# B&R Automation Studio project TD52 (part 43)

#### c_parCyclic.st
```iecst
(*******************************************************************************
CUSTOMIZED: c_par 			customized reserve parameters 1-200

This code is confidential and proprietary to the INNIO Company.
It may not be used in any form, or reproduced in any manner,
without written permission of the INNIO Company.
Copyright, INNIO Company, 2019

Customized modifications: -
------------------------

History:
-------
V3.20.0	02.03.2011 lettenb.	new, old default-settings removed
...
V4.00.0	08.05.2014 Zengerer ?hit? to int with optional factory default values
V4.02.0 24.06.2015 Zengerer cleanup
V4.04.0	20.06.2016 Weitzer	add reserve parameter 71..200
V4.11.0	31.01.2022 Zengerer	array preparation for import HMI Extensions 201..500

Instructions for use:
--------------------
- define customized use of reserve parameters here
- mark used channels here, to avoid duplicate usage withhin one customer project

AVOID HARDCODED Para.xxx VALUES!
You MAYBE want to enter SOME factory default values, but ONLY TO THE Para_FactoryDefault.xxx STRUCTURE!
By this way the parameter values in Para.xxx would stay acessible according to XT4 parameter management process.

***********************************************
further use for TP only!
***********************************************

Outstandings:
------------
	Para.iCtr_Mns_Options := REAL_TO_INT(Para.rCust_SparePara[72]) ;		ToDO: remove, when parameter gets availabel on VIS

*******************************************************************************)
PROGRAM _CYCLIC

	Para.rCust_SparePara[1]	;	(*MARK USAGE HERE, to avoid duplicate usage*)	(*  =   SPS_REZP1 *)
	OUT_CU.rCust_SparePara[1];	(*para values get copied to module OUT interface, to allow possible usage in other modules also. Edit other´s module .vvm accordingly, if needed. *)

	Para.rCust_SparePara[2]	; 													(*  =   SPS_REZP2 *)
	OUT_CU.rCust_SparePara[2];													(*  =	SPS_REZP2 *)

	Para.rCust_SparePara[3]	;  													(*  =	SPS_REZP3 *)
	OUT_CU.rCust_SparePara[3];													(*  =	SPS_REZP3 *)

	Para.rCust_SparePara[4]	;													(*  =   SPS_REZP4*)
	OUT_CU.rCust_SparePara[4];													(*  =	SPS_REZP4 *)

	Para.rCust_SparePara[5]	; 													(*  =   SPS_REZP5*)
	OUT_CU.rCust_SparePara[5];													(*  =	SPS_REZP5 *)

	Para.rCust_SparePara[6]	;  													(*  =	SPS_REZP6*)
	OUT_CU.rCust_SparePara[6];													(*  =	SPS_REZP6 *)

	Para.rCust_SparePara[7]	;  													(*  =	SPS_REZP7*)
	OUT_CU.rCust_SparePara[7] ;													(*  =	SPS_REZP7 *)

	Para.rCust_SparePara[8]	;   												(*  =	SPS_REZP8*)
	OUT_CU.rCust_SparePara[8] ;													(*  =	SPS_REZP8 *)

	Para.rCust_SparePara[9]		;  												(*  =	SPS_REZP9*)
	OUT_CU.rCust_SparePara[9] 	;												(*  =	SPS_REZP9 *)

	Para.rCust_SparePara[10]	;  												(*  =	SPS_REZP10*)
	OUT_CU.rCust_SparePara[10]	;												(*  =	SPS_REZP10 *)

	(*------------------------------------------------------------------*)
	Para.rCust_SparePara[11] 	;	(*  =	SPS_REZP11 *)
	OUT_CU.rCust_SparePara[11]	;	(*  =	SPS_REZP11 *)

	Para.rCust_SparePara[12]	;	(*  =	SPS_REZP12 *)
	OUT_CU.rCust_SparePara[12]	;	(*  =	SPS_REZP12 *)

	Para.rCust_SparePara[13]	;	(*  =	SPS_REZP13 *)
	OUT_CU.rCust_SparePara[13]	;	(*  =	SPS_REZP13 *)

	Para.rCust_SparePara[14]	;	(*  =	SPS_REZP14 *)
	OUT_CU.rCust_SparePara[14]	;	(*  =	SPS_REZP14 *)

	Para.rCust_SparePara[15]	;	(*  =	SPS_REZP15 *)
	OUT_CU.rCust_SparePara[15]	;	(*  =	SPS_REZP15 *)

	Para.rCust_SparePara[16]	;	(*  =	SPS_REZP16 *)
	OUT_CU.rCust_SparePara[16]	;	(*  =	SPS_REZP16 *)

	Para.rCust_SparePara[17]	;	(*  =	SPS_REZP17 *)
	OUT_CU.rCust_SparePara[17]	;	(*  =	SPS_REZP17 *)

	Para.rCust_SparePara[18]	;	(*  =	SPS_REZP18 *)
	OUT_CU.rCust_SparePara[18]	;	(*  =	SPS_REZP18 *)

	Para.rCust_SparePara[19]	;	(*  =	SPS_REZP19 *)
	OUT_CU.rCust_SparePara[19]	;	(*  =	SPS_REZP19 *)

	Para.rCust_SparePara[20]	;	(*  =	SPS_REZP20 *)
	OUT_CU.rCust_SparePara[20]	;	(*  =	SPS_REZP20 *)

	(*------------------------------------------------------------------*)
	Para.rCust_SparePara[21]	;	(*  =	SPS_REZP21*)
	OUT_CU.rCust_SparePara[21] ;	(*  =	SPS_REZP21; *)

	Para.rCust_SparePara[22]	;	(*  =	SPS_REZP22*)
	OUT_CU.rCust_SparePara[22] ;	(*  =	SPS_REZP22; *)

	Para.rCust_SparePara[23]	;	(*  =	SPS_REZP23*)
	OUT_CU.rCust_SparePara[23] ;	(*  =	SPS_REZP23; *)

	Para.rCust_SparePara[24]	;	(*  =	SPS_REZP24*)
	OUT_CU.rCust_SparePara[24] ;	(*  =	SPS_REZP24; *)

	Para.rCust_SparePara[25]	;	(*  =	SPS_REZP25*)
	OUT_CU.rCust_SparePara[25] ;	(*  =	SPS_REZP25; *)

	Para.rCust_SparePara[26]	;	(*  =	SPS_REZP26*)
	OUT_CU.rCust_SparePara[26] ;	(*  =	SPS_REZP26; *)

	Para.rCust_SparePara[27]	;	(*  =	SPS_REZP27*)
	OUT_CU.rCust_SparePara[27] ;	(*  =	SPS_REZP27; *)

	Para.rCust_SparePara[28]	;	(*  =	SPS_REZP28*)
	OUT_CU.rCust_SparePara[28] ;	(*  =	SPS_REZP28; *)

	Para.rCust_SparePara[29]	;	(*  =	SPS_REZP29*)
	OUT_CU.rCust_SparePara[29] ;	(*  =	SPS_REZP29; *)

	OUT_CU.rCust_SparePara[30] ;	(*  =	SPS_REZP30; *)

	(*------------------------------------------------------------------*)
	Para.rCust_SparePara[31]	;	(*  =	SPS_REZP31*)
	OUT_CU.rCust_SparePara[31] ;	(*  =	SPS_REZP31; *)

	Para.rCust_SparePara[32]	;	(*  =	SPS_REZP32*)
	OUT_CU.rCust_SparePara[32] ;	(*  =	SPS_REZP32; *)

	Para.rCust_SparePara[33]	;	(*  =	SPS_REZP33*)
	OUT_CU.rCust_SparePara[33] ;	(*  =	SPS_REZP33; *)

	Para.rCust_SparePara[34]	;	(*  =	SPS_REZP34*)
	OUT_CU.rCust_SparePara[34] ;	(*  =	SPS_REZP34; *)

	Para.rCust_SparePara[35]	;	(*  =	SPS_REZP35*)
	OUT_CU.rCust_SparePara[35] ;	(*  =	SPS_REZP35; *)

	Para.rCust_SparePara[36]	;	(*  =	SPS_REZP36*)
	OUT_CU.rCust_SparePara[36] ;	(*  =	SPS_REZP36; *)

	Para.rCust_SparePara[37]	;	(*  =	SPS_REZP37*)
	OUT_CU.rCust_SparePara[37] ;	(*  =	SPS_REZP37; *)

	Para.rCust_SparePara[38]	;	(*  =	SPS_REZP38*)
	OUT_CU.rCust_SparePara[38] ;	(*  =	SPS_REZP38; *)

	Para.rCust_SparePara[39]	;	(*  =	SPS_REZP39*)
	OUT_CU.rCust_SparePara[39] ;	(*  =	SPS_REZP39; *)

	Para.rCust_SparePara[40]	;	(*  =	SPS_REZP40*)
	OUT_CU.rCust_SparePara[40] ;	(*  =	SPS_REZP40; *)

	(*------------------------------------------------------------------*)
	Para.rCust_SparePara[41]	;	(*  =	SPS_REZP41*)
	OUT_CU.rCust_SparePara[41] ;	(*  =	SPS_REZP41; *)

	Para.rCust_SparePara[42]	;	(*  =	SPS_REZP42*)
	OUT_CU.rCust_SparePara[42] ;	(*  =	SPS_REZP42; *)

	Para.rCust_SparePara[43]	;	(*  =	SPS_REZP43*)
	OUT_CU.rCust_SparePara[43] ;	(*  =	SPS_REZP43; *)

	Para.rCust_SparePara[44]	;	(*  =	SPS_REZP44*)
	OUT_CU.rCust_SparePara[44] ;	(*  =	SPS_REZP44; *)

	Para.rCust_SparePara[45]	;	(*  =	SPS_REZP45*)
	OUT_CU.rCust_SparePara[45] ;	(*  =	SPS_REZP45; *)

	Para.rCust_SparePara[46]	;	(*  =	SPS_REZP46*)
	OUT_CU.rCust_SparePara[46] ;	(*  =	SPS_REZP46; *)

	Para.rCust_SparePara[47]	;	(*  =	SPS_REZP47*)
	OUT_CU.rCust_SparePara[47] ;	(*  =	SPS_REZP47; *)

	Para.rCust_SparePara[48]	;	(*  =	SPS_REZP48*)
	OUT_CU.rCust_SparePara[48] ;	(*  =	SPS_REZP48; *)

	Para.rCust_SparePara[49]	;	(*  =	SPS_REZP49*)
	OUT_CU.rCust_SparePara[49] ;	(*  =	SPS_REZP49; *)

	Para.rCust_SparePara[50]	;	(*  =	SPS_REZP50*)
	OUT_CU.rCust_SparePara[50] ;	(*  =	SPS_REZP50; *)

	(*------------------------------------------------------------------*)
	Para.rCust_SparePara[51]	;	(*  =	SPS_REZP51*)
	OUT_CU.rCust_SparePara[51] ;	(*  =	SPS_REZP51; *)

	Para.rCust_SparePara[52]	;	(*  =	SPS_REZP52*)
	OUT_CU.rCust_SparePara[52] ;	(*  =	SPS_REZP52; *)

	Para.rCust_SparePara[53]	;	(*  =	SPS_REZP53*)
	OUT_CU.rCust_SparePara[53] ;	(*  =	SPS_REZP53; *)

	Para.rCust_SparePara[54]	;	(*  =	SPS_REZP54*)
	OUT_CU.rCust_SparePara[54] ;	(*  =	SPS_REZP54; *)

	Para.rCust_SparePara[55]	;	(*  =	SPS_REZP55*)
	OUT_CU.rCust_SparePara[55] ;	(*  =	SPS_REZP55; *)

	Para.rCust_SparePara[56]	;	(*  =	SPS_REZP56*)
	OUT_CU.rCust_SparePara[56] ;	(*  =	SPS_REZP56; *)

	Para.rCust_SparePara[57]	;	(*  =	SPS_REZP57*)
	OUT_CU.rCust_SparePara[57] ;	(*  =	SPS_REZP57; *)

	Para.rCust_SparePara[58]	;	(*  =	SPS_REZP58*)
	OUT_CU.rCust_SparePara[58] ;	(*  =	SPS_REZP58; *)

	Para.rCust_SparePara[59]	;	(*  =	SPS_REZP59*)
	OUT_CU.rCust_SparePara[59] ;	(*  =	SPS_REZP59; *)

	Para.rCust_SparePara[60]	;	(*  =	SPS_REZP60*)
	OUT_CU.rCust_SparePara[60] ;	(*  =	SPS_REZP60; *)

	(*------------------------------------------------------------------*)
	Para.rCust_SparePara[61]	;	(*  =	SPS_REZP61*)
	OUT_CU.rCust_SparePara[61] ;	(* = 	ssResPara61 *)

	Para.rCust_SparePara[62]	;	(*  =	SPS_REZP62*)
	OUT_CU.rCust_SparePara[62] ;	(* = 	ssResPara62 *)

	Para.rCust_SparePara[63]	;	(*  =	SPS_REZP63*)
	OUT_CU.rCust_SparePara[63] ;	(* = 	ssResPara63 *)

	Para.rCust_SparePara[64]	;	(*  =	SPS_REZP64*)
	OUT_CU.rCust_SparePara[64] ;	(* = 	ssResPara64 *)

	Para.rCust_SparePara[65]	;	(*  =	SPS_REZP65*)
	OUT_CU.rCust_SparePara[65] ;	(* = 	ssResPara65 *)

	Para.rCust_SparePara[66]	;	(*  =	SPS_REZP66*)
	OUT_CU.rCust_SparePara[66] ;	(* = 	ssResPara66 *)

	Para.rCust_SparePara[67]	;	(*  =	SPS_REZP67*)
	OUT_CU.rCust_SparePara[67] ;	(* = 	ssResPara67 *)

	Para.rCust_SparePara[68]	;	(*  =	SPS_REZP68*)
	OUT_CU.rCust_SparePara[68] ;	(* = 	ssResPara68 *)

	Para.rCust_SparePara[69]	;	(*  =	SPS_REZP69 *)
	OUT_CU.rCust_SparePara[69] ;	(* = 	ssResPara69 *)

	Para.rCust_SparePara[70]	;	(*  =	SPS_REZP70 *)
	OUT_CU.rCust_SparePara[70] ;	(* = 	ssResPara70 *)

	(*---------------------------------------------------------------------------------------*)
	(* END OF PRECONFIGURED VISUALISATION DATA POINS on standard engines, up to Vis Rev. 4.x *)
	(*---------------------------------------------------------------------------------------*)
	Para.rCust_SparePara[71];		(*  = SPS_REZP	71	***USED*** *)
	OUT_CU.rCust_SparePara[71];		(*  = ssResPara	71	*)

	Para.rCust_SparePara[72];		(*  = SPS_REZP	72  ***USED*** *)
	OUT_CU.rCust_SparePara[72];		(*  = ssResPara	72	*)

	Para.rCust_SparePara[73];		(*  = SPS_REZP	73	***USED*** *)
	OUT_CU.rCust_SparePara[73];		(*  = ssResPara	73	*)

	Para.rCust_SparePara[74];		(*  = SPS_REZP	74	*)
	OUT_CU.rCust_SparePara[74];		(*  = ssResPara	74	*)

	Para.rCust_SparePara[75];		(*  = SPS_REZP	75	*)
	OUT_CU.rCust_SparePara[75];		(*  = ssResPara	75	*)

	Para.rCust_SparePara[76];		(*  = SPS_REZP	76	*)
	OUT_CU.rCust_SparePara[76];		(*  = ssResPara	76	*)

	Para.rCust_SparePara[77];		(*  = SPS_REZP	77	*)
	OUT_CU.rCust_SparePara[77];		(*  = ssResPara	77	*)

	Para.rCust_SparePara[78];		(*  = SPS_REZP	78	*)
	OUT_CU.rCust_SparePara[78];		(*  = ssResPara	78	*)

	Para.rCust_SparePara[79];		(*  = SPS_REZP	79	*)
	OUT_CU.rCust_SparePara[79];		(*  = ssResPara	79	*)

	Para.rCust_SparePara[80];		(*  = SPS_REZP	80	*)
	OUT_CU.rCust_SparePara[80];		(*  = ssResPara	80	*)

	(*------------------------------------------------------------------*)
	Para.rCust_SparePara[81];		(*  = SPS_REZP	81	*)
	OUT_CU.rCust_SparePara[81];		(*  = ssResPara	81	*)

	Para.rCust_SparePara[82];		(*  = SPS_REZP	82	*)
	OUT_CU.rCust_SparePara[82];		(*  = ssResPara	82	*)

	Para.rCust_SparePara[83];		(*  = SPS_REZP	83	*)
	OUT_CU.rCust_SparePara[83];		(*  = ssResPara	83	*)

	Para.rCust_SparePara[84];		(*  = SPS_REZP	84	*)
	OUT_CU.rCust_SparePara[84];		(*  = ssResPara	84	*)

	Para.rCust_SparePara[85];		(*  = SPS_REZP	85	*)
	OUT_CU.rCust_SparePara[85];		(*  = ssResPara	85	*)

	Para.rCust_SparePara[86];		(*  = SPS_REZP	86	*)
	OUT_CU.rCust_SparePara[86];		(*  = ssResPara	86	*)

	Para.rCust_SparePara[87];		(*  = SPS_REZP	87	*)
	OUT_CU.rCust_SparePara[87];		(*  = ssResPara	87	*)

	Para.rCust_SparePara[88];		(*  = SPS_REZP	88	*)
	OUT_CU.rCust_SparePara[88];		(*  = ssResPara	88	*)

	Para.rCust_SparePara[89];		(*  = SPS_REZP	89	*)
	OUT_CU.rCust_SparePara[89];		(*  = ssResPara	89	*)

	Para.rCust_SparePara[90];		(*  = SPS_REZP	90	*)
	OUT_CU.rCust_SparePara[90];		(*  = ssResPara	90	*)

	(*------------------------------------------------------------------*)
	Para.rCust_SparePara[91];		(*  = SPS_REZP	91	*)
	OUT_CU.rCust_SparePara[91];		(*  = ssResPara	91	*)

	Para.rCust_SparePara[92];		(*  = SPS_REZP	92	*)
	OUT_CU.rCust_SparePara[92];		(*  = ssResPara	92	*)

	Para.rCust_SparePara[93];		(*  = SPS_REZP	93	*)
	OUT_CU.rCust_SparePara[93];		(*  = ssResPara	93	*)

	Para.rCust_SparePara[94];		(*  = SPS_REZP	94	*)
	OUT_CU.rCust_SparePara[94];		(*  = ssResPara	94	*)

	Para.rCust_SparePara[95];		(*  = SPS_REZP	95	*)
	OUT_CU.rCust_SparePara[95];		(*  = ssResPara	95	*)

	Para.rCust_SparePara[96];		(*  = SPS_REZP	96	*)
	OUT_CU.rCust_SparePara[96];		(*  = ssResPara	96	*)

	Para.rCust_SparePara[97];		(*  = SPS_REZP	97	*)
	OUT_CU.rCust_SparePara[97];		(*  = ssResPara	97	*)

	Para.rCust_SparePara[98];		(*  = SPS_REZP	98	*)
	OUT_CU.rCust_SparePara[98];		(*  = ssResPara	98	*)

	Para.rCust_SparePara[99];		(*  = SPS_REZP	99	*)
	OUT_CU.rCust_SparePara[99];		(*  = ssResPara	99	*)

	Para.rCust_SparePara[100];		(*  = SPS_REZP	100	*)
	OUT_CU.rCust_SparePara[100];	(*  = ssResPara	100	*)

	(*------------------------------------------------------------------*)
	Para.rCust_SparePara[101];		(*  = SPS_REZP	101	*)
	OUT_CU.rCust_SparePara[101];	(*  = ssResPara	101	*)

	Para.rCust_SparePara[102];		(*  = SPS_REZP	102	*)
	OUT_CU.rCust_SparePara[102];	(*  = ssResPara	102	*)

	Para.rCust_SparePara[103];		(*  = SPS_REZP	103	*)
	OUT_CU.rCust_SparePara[103];	(*  = ssResPara	103	*)

	Para.rCust_SparePara[104];		(*  = SPS_REZP	104	*)
	OUT_CU.rCust_SparePara[104];	(*  = ssResPara	104	*)

	Para.rCust_SparePara[105];		(*  = SPS_REZP	105	*)
	OUT_CU.rCust_SparePara[105];	(*  = ssResPara	105	*)

	Para.rCust_SparePara[106];		(*  = SPS_REZP	106	*)
	OUT_CU.rCust_SparePara[106];	(*  = ssResPara	106	*)

	Para.rCust_SparePara[107];		(*  = SPS_REZP	107	*)
	OUT_CU.rCust_SparePara[107];	(*  = ssResPara	107	*)

	Para.rCust_SparePara[108];		(*  = SPS_REZP	108	*)
	OUT_CU.rCust_SparePara[108];	(*  = ssResPara	108	*)

	Para.rCust_SparePara[109];		(*  = SPS_REZP	109	*)
	OUT_CU.rCust_SparePara[109];	(*  = ssResPara	109	*)

	Para.rCust_SparePara[110];		(*  = SPS_REZP	110	*)
	OUT_CU.rCust_SparePara[110];	(*  = ssResPara	110	*)

	(*------------------------------------------------------------------*)
	Para.rCust_SparePara[111];		(*  = SPS_REZP	111	*)
	OUT_CU.rCust_SparePara[111];	(*  = ssResPara	111	*)

	Para.rCust_SparePara[112];		(*  = SPS_REZP	112	*)
	OUT_CU.rCust_SparePara[112];	(*  = ssResPara	112	*)

	Para.rCust_SparePara[113];		(*  = SPS_REZP	113	*)
	OUT_CU.rCust_SparePara[113];	(*  = ssResPara	113	*)

	Para.rCust_SparePara[114];		(*  = SPS_REZP	114	*)
	OUT_CU.rCust_SparePara[114];	(*  = ssResPara	114	*)

	Para.rCust_SparePara[115];		(*  = SPS_REZP	115	*)
	OUT_CU.rCust_SparePara[115];	(*  = ssResPara	115	*)

	Para.rCust_SparePara[116];		(*  = SPS_REZP	116	*)
	OUT_CU.rCust_SparePara[116];	(*  = ssResPara	116	*)

	Para.rCust_SparePara[117];		(*  = SPS_REZP	117	*)
	OUT_CU.rCust_SparePara[117];	(*  = ssResPara	117	*)

	Para.rCust_SparePara[118];		(*  = SPS_REZP	118	*)
	OUT_CU.rCust_SparePara[118];	(*  = ssResPara	118	*)

	Para.rCust_SparePara[119];		(*  = SPS_REZP	119	*)
	OUT_CU.rCust_SparePara[119];	(*  = ssResPara	119	*)

	Para.rCust_SparePara[120];		(*  = SPS_REZP	120	*)
	OUT_CU.rCust_SparePara[120];	(*  = ssResPara	120	*)

	(*------------------------------------------------------------------*)
	Para.rCust_SparePara[121];		(*  = SPS_REZP	121	*)
	OUT_CU.rCust_SparePara[121];	(*  = ssResPara	121	*)

	Para.rCust_SparePara[122];		(*  = SPS_REZP	122	*)
	OUT_CU.rCust_SparePara[122];	(*  = ssResPara	122	*)

	Para.rCust_SparePara[123];		(*  = SPS_REZP	123	*)
	OUT_CU.rCust_SparePara[123];	(*  = ssResPara	123	*)

	Para.rCust_SparePara[124];		(*  = SPS_REZP	124	*)
	OUT_CU.rCust_SparePara[124];	(*  = ssResPara	124	*)

	Para.rCust_SparePara[125];		(*  = SPS_REZP	125	*)
	OUT_CU.rCust_SparePara[125];	(*  = ssResPara	125	*)

	Para.rCust_SparePara[126];		(*  = SPS_REZP	126	*)
	OUT_CU.rCust_SparePara[126];	(*  = ssResPara	126	*)

	Para.rCust_SparePara[127];		(*  = SPS_REZP	127	*)
	OUT_CU.rCust_SparePara[127];	(*  = ssResPara	127	*)

	Para.rCust_SparePara[128];		(*  = SPS_REZP	128	*)
	OUT_CU.rCust_SparePara[128];	(*  = ssResPara	128	*)

	Para.rCust_SparePara[129];		(*  = SPS_REZP	129	*)
	OUT_CU.rCust_SparePara[129];	(*  = ssResPara	129	*)

	Para.rCust_SparePara[130];		(*  = SPS_REZP	130	*)
	OUT_CU.rCust_SparePara[130];	(*  = ssResPara	130	*)

	(*------------------------------------------------------------------*)
	Para.rCust_SparePara[131];		(*  = SPS_REZP	131	*)
	OUT_CU.rCust_SparePara[131];	(*  = ssResPara	131	*)

	Para.rCust_SparePara[132];		(*  = SPS_REZP	132	*)
	OUT_CU.rCust_SparePara[132];	(*  = ssResPara	132	*)

	Para.rCust_SparePara[133];		(*  = SPS_REZP	133	*)
	OUT_CU.rCust_SparePara[133];	(*  = ssResPara	133	*)

	Para.rCust_SparePara[134];		(*  = SPS_REZP	134	*)
	OUT_CU.rCust_SparePara[134];	(*  = ssResPara	134	*)

	Para.rCust_SparePara[135];		(*  = SPS_REZP	135	*)
	OUT_CU.rCust_SparePara[135];	(*  = ssResPara	135	*)

	Para.rCust_SparePara[136];		(*  = SPS_REZP	136	*)
	OUT_CU.rCust_SparePara[136];	(*  = ssResPara	136	*)

	Para.rCust_SparePara[137];		(*  = SPS_REZP	137	*)
	OUT_CU.rCust_SparePara[137];	(*  = ssResPara	137	*)

	Para.rCust_SparePara[138];		(*  = SPS_REZP	138	*)
	OUT_CU.rCust_SparePara[138];	(*  = ssResPara	138	*)

	Para.rCust_SparePara[139];		(*  = SPS_REZP	139	*)
	OUT_CU.rCust_SparePara[139];	(*  = ssResPara	139	*)

	Para.rCust_SparePara[140];		(*  = SPS_REZP	140	*)
	OUT_CU.rCust_SparePara[140];	(*  = ssResPara	140	*)

	(*------------------------------------------------------------------*)
	Para.rCust_SparePara[141];		(*  = SPS_REZP	141	*)
	OUT_CU.rCust_SparePara[141];	(*  = ssResPara	141	*)

	Para.rCust_SparePara[142];		(*  = SPS_REZP	142	*)
	OUT_CU.rCust_SparePara[142];	(*  = ssResPara	142	*)

	Para.rCust_SparePara[143];		(*  = SPS_REZP	143	*)
	OUT_CU.rCust_SparePara[143];	(*  = ssResPara	143	*)

	Para.rCust_SparePara[144];		(*  = SPS_REZP	144	*)
	OUT_CU.rCust_SparePara[144];	(*  = ssResPara	144	*)

	Para.rCust_SparePara[145];		(*  = SPS_REZP	145	*)
	OUT_CU.rCust_SparePara[145];	(*  = ssResPara	145	*)

	Para.rCust_SparePara[146];		(*  = SPS_REZP	146	*)
	OUT_CU.rCust_SparePara[146];	(*  = ssResPara	146	*)

	Para.rCust_SparePara[147];		(*  = SPS_REZP	147	*)
	OUT_CU.rCust_SparePara[147];	(*  = ssResPara	147	*)

	Para.rCust_SparePara[148];		(*  = SPS_REZP	148	*)
	OUT_CU.rCust_SparePara[148];	(*  = ssResPara	148	*)

	Para.rCust_SparePara[149];		(*  = SPS_REZP	149	*)
	OUT_CU.rCust_SparePara[149];	(*  = ssResPara	149	*)

	Para.rCust_SparePara[150];		(*  = SPS_REZP	150	*)
	OUT_CU.rCust_SparePara[150];	(*  = ssResPara	150	*)

	(*------------------------------------------------------------------*)
	Para.rCust_SparePara[151];		(*  = SPS_REZP	151	*)
	OUT_CU.rCust_SparePara[151];	(*  = ssResPara	151	*)

	Para.rCust_SparePara[152];		(*  = SPS_REZP	152	*)
	OUT_CU.rCust_SparePara[152];	(*  = ssResPara	152	*)

	Para.rCust_SparePara[153];		(*  = SPS_REZP	153	*)
	OUT_CU.rCust_SparePara[153];	(*  = ssResPara	153	*)

	Para.rCust_SparePara[154];		(*  = SPS_REZP	154	*)
	OUT_CU.rCust_SparePara[154];	(*  = ssResPara	154	*)

	Para.rCust_SparePara[155];		(*  = SPS_REZP	155	*)
	OUT_CU.rCust_SparePara[155];	(*  = ssResPara	155	*)

	Para.rCust_SparePara[156];		(*  = SPS_REZP	156	*)
	OUT_CU.rCust_SparePara[156];	(*  = ssResPara	156	*)

	Para.rCust_SparePara[157];		(*  = SPS_REZP	157	*)
	OUT_CU.rCust_SparePara[157];	(*  = ssResPara	157	*)

	Para.rCust_SparePara[158];		(*  = SPS_REZP	158	*)
	OUT_CU.rCust_SparePara[158];	(*  = ssResPara	158	*)

	Para.rCust_SparePara[159];		(*  = SPS_REZP	159	*)
	OUT_CU.rCust_SparePara[159];	(*  = ssResPara	159	*)

	Para.rCust_SparePara[160];		(*  = SPS_REZP	160	*)
	OUT_CU.rCust_SparePara[160];	(*  = ssResPara	160	*)

	(*------------------------------------------------------------------*)
	Para.rCust_SparePara[161];		(*  = SPS_REZP	161	*)
	OUT_CU.rCust_SparePara[161];	(*  = ssResPara	161	*)

	Para.rCust_SparePara[162];		(*  = SPS_REZP	162	*)
	OUT_CU.rCust_SparePara[162];	(*  = ssResPara	162	*)

	Para.rCust_SparePara[163];		(*  = SPS_REZP	163	*)
	OUT_CU.rCust_SparePara[163];	(*  = ssResPara	163	*)

	Para.rCust_SparePara[164];		(*  = SPS_REZP	164	*)
	OUT_CU.rCust_SparePara[164];	(*  = ssResPara	164	*)

	Para.rCust_SparePara[165];		(*  = SPS_REZP	165	*)
	OUT_CU.rCust_SparePara[165];	(*  = ssResPara	165	*)

	Para.rCust_SparePara[166];		(*  = SPS_REZP	166	*)
	OUT_CU.rCust_SparePara[166];	(*  = ssResPara	166	*)

	Para.rCust_SparePara[167];		(*  = SPS_REZP	167	*)
	OUT_CU.rCust_SparePara[167];	(*  = ssResPara	167	*)

	Para.rCust_SparePara[168];		(*  = SPS_REZP	168	*)
	OUT_CU.rCust_SparePara[168];	(*  = ssResPara	168	*)

	Para.rCust_SparePara[169];		(*  = SPS_REZP	169	*)
	OUT_CU.rCust_SparePara[169];	(*  = ssResPara	169	*)

	Para.rCust_SparePara[170];		(*  = SPS_REZP	170	*)
	OUT_CU.rCust_SparePara[170];	(*  = ssResPara	170	*)

	(*------------------------------------------------------------------*)
	Para.rCust_SparePara[171];		(*  = SPS_REZP	171	*)
	OUT_CU.rCust_SparePara[171];	(*  = ssResPara	171	*)

	Para.rCust_SparePara[172];		(*  = SPS_REZP	172	*)
	OUT_CU.rCust_SparePara[172];	(*  = ssResPara	172	*)

	Para.rCust_SparePara[173];		(*  = SPS_REZP	173	*)
	OUT_CU.rCust_SparePara[173];	(*  = ssResPara	173	*)

	Para.rCust_SparePara[174];		(*  = SPS_REZP	174	*)
	OUT_CU.rCust_SparePara[174];	(*  = ssResPara	174	*)

	Para.rCust_SparePara[175];		(*  = SPS_REZP	175	*)
	OUT_CU.rCust_SparePara[175];	(*  = ssResPara	175	*)

	Para.rCust_SparePara[176];		(*  = SPS_REZP	176	*)
	OUT_CU.rCust_SparePara[176];	(*  = ssResPara	176	*)

	Para.rCust_SparePara[177];		(*  = SPS_REZP	177	*)
	OUT_CU.rCust_SparePara[177];	(*  = ssResPara	177	*)

	Para.rCust_SparePara[178];		(*  = SPS_REZP	178	*)
	OUT_CU.rCust_SparePara[178];	(*  = ssResPara	178	*)

	Para.rCust_SparePara[179];		(*  = SPS_REZP	179	*)
	OUT_CU.rCust_SparePara[179];	(*  = ssResPara	179	*)

	Para.rCust_SparePara[180];		(*  = SPS_REZP	180	*)
	OUT_CU.rCust_SparePara[180];	(*  = ssResPara	180	*)

	(*------------------------------------------------------------------*)
	Para.rCust_SparePara[181];		(*  = SPS_REZP	181	*)
	OUT_CU.rCust_SparePara[181];	(*  = ssResPara	181	*)

	Para.rCust_SparePara[182];		(*  = SPS_REZP	182	*)
	OUT_CU.rCust_SparePara[182];	(*  = ssResPara	182	*)

	Para.rCust_SparePara[183];		(*  = SPS_REZP	183	*)
	OUT_CU.rCust_SparePara[183];	(*  = ssResPara	183	*)

	Para.rCust_SparePara[184];		(*  = SPS_REZP	184	*)
	OUT_CU.rCust_SparePara[184];	(*  = ssResPara	184	*)

	Para.rCust_SparePara[185];		(*  = SPS_REZP	185	*)
	OUT_CU.rCust_SparePara[185];	(*  = ssResPara	185	*)

	Para.rCust_SparePara[186];		(*  = SPS_REZP	186	*)
	OUT_CU.rCust_SparePara[186];	(*  = ssResPara	186	*)

	Para.rCust_SparePara[187];		(*  = SPS_REZP	187	*)
	OUT_CU.rCust_SparePara[187];	(*  = ssResPara	187	*)

	Para.rCust_SparePara[188];		(*  = SPS_REZP	188	*)
	OUT_CU.rCust_SparePara[188];	(*  = ssResPara	188	*)

	Para.rCust_SparePara[189];		(*  = SPS_REZP	189	*)
	OUT_CU.rCust_SparePara[189];	(*  = ssResPara	189	*)

	Para.rCust_SparePara[190];		(*  = SPS_REZP	190	*)
	OUT_CU.rCust_SparePara[190];	(*  = ssResPara	190	*)

	(*------------------------------------------------------------------*)
	Para.rCust_SparePara[191];		(*  = SPS_REZP	191	*)
	OUT_CU.rCust_SparePara[191];	(*  = ssResPara	191	*)

	Para.rCust_SparePara[192];		(*  = SPS_REZP	192	*)
	OUT_CU.rCust_SparePara[192];	(*  = ssResPara	192	*)

	Para.rCust_SparePara[193];		(*  = SPS_REZP	193	*)
	OUT_CU.rCust_SparePara[193];	(*  = ssResPara	193	*)

	Para.rCust_SparePara[194];		(*  = SPS_REZP	194	*)
	OUT_CU.rCust_SparePara[194];	(*  = ssResPara	194	*)

	Para.rCust_SparePara[195];		(*  = SPS_REZP	195	*)
	OUT_CU.rCust_SparePara[195];	(*  = ssResPara	195	*)

	Para.rCust_SparePara[196];		(*  = SPS_REZP	196	*)
	OUT_CU.rCust_SparePara[196];	(*  = ssResPara	196	*)

	Para.rCust_SparePara[197];		(*  = SPS_REZP	197	*)
	OUT_CU.rCust_SparePara[197];	(*  = ssResPara	197	*)

	Para.rCust_SparePara[198];		(*  = SPS_REZP	198	*)
	OUT_CU.rCust_SparePara[198];	(*  = ssResPara	198	*)

	Para.rCust_SparePara[199];		(*  = SPS_REZP	199	*)
	OUT_CU.rCust_SparePara[199];	(*  = ssResPara	199	*)

	Para.rCust_SparePara[200];		(*  = SPS_REZP	200	*)
	OUT_CU.rCust_SparePara[200];	(*  = ssResPara	200	*)

	(*------------------------------------------------------------------*)

	(***********************************************
	END OF CONFIGURATION AREA
	***********************************************)
	(* NO CHANGES BEJOND THIS LINE! *)

//	OUT_CU.rCust_SparePara := 		Para.rCust_SparePara     ;	(* DONT DO THIS ANY MORE since different array size is possible with HMI Extention import in V4.11  *)
	iOut_SparePara_Size := SIZEOF(OUT_CU.rCust_SparePara)/ SIZEOF(OUT_CU.rCust_SparePara[0]) -1 ;
	FOR n := 0 TO iOut_SparePara_Size DO
		OUT_CU.rCust_SparePara[n] := 		Para.rCust_SparePara[n]     ;	(* Copy all parameter values to Module OUT interface for possible reuse in other modules  *)
	END_FOR

END_PROGRAM
```

#### c_par.var
```iecst
VAR
	iOut_SparePara_Size : UDINT := 0;
	n : UDINT := 0;
END_VAR
```

### Program Logical/Customized/c_ctr (IEC, version 4.11.0) - Interface connection for  customizable controllers

#### c_ctrCyclic.st - Cyclic code
```iecst
(*******************************************************************************
CUSTOMIZED: c_ctr 		reserve controller handling (cyclic)

This code is confidential AND proprietary to the INNIO Company.
It may NOT be used in any form, or reproduced in any manner,
without written permission of the INNIO Company.
Copyright, INNIO Company, 2022

Customized modifications: -
------------------------

History:
-------
		23.05.2012	Zengerer	generated, new
V4.02	09.09.2015	Zengerer	cleanup, prototype entry FOR documentation comments
V4.04	20.06.2016	Weitzer		add controller 41 .. 45
V4.05	23.01.2018	Perktold	added option for humitity control with ctr. 2
V4.11	27.01.2022	Perktold	impemented plant controller upgrade (2nd W_set, Gain Scheduling, Retrigger, cust. Ymin/max)
		31.01.2022	zengerer	extended controller items 41-45 ONLY FOR USE WITH HMI Extension Package!

Instructions FOR use:
--------------------
-
Outstandings:
------------
- ENTFERNEN: IF NOT bEnableTestBench THEN   (*NUR FÜR TPSS- Prüfstand...

*******************************************************************************)

PROGRAM _CYCLIC
																																		//	IF NOT bEnableTestBench THEN   (*Bit bEnableTestBench NUR FÜR TP- Prüfstand aktivieren*)

	(* customizable controller X 		*** PROTOTYPE EXAMPLE ***
	VIS2MM.tCtr_Cust1_In.enable			:= Para.bCtr_Cust1 AND TRUE;	* enable controller with parameter / AND connect additional enable bits here *
	VIS2MM.tCtr_Cust1_In.X				:= 0;							* connect actual controller value here  *
	VIS2MM.tCtr_Cust1_In.W_ext			:= 0;							* optional: connect external controller setpoint value here  *
	VIS2MM.tCtr_Cust1_In.W_ext_Active	:= FALSE;						* optional: connect activation of external setpoint here  *
	VIS2MM.tCtr_Cust1_In.W_set2_Active	:= FALSE;						* optional: connect signal to switch to 2nd internal setpoint here  *
	VIS2MM.tCtr_Cust1_In.GainScheduling	:= 0.0;							* optional: connect Gain Scheduling signal here, limits [0.0-1.0] : 0.0 = use 100% of the standard PID-parameters | 1.0 = use 100% of the GainSched. PID Parameters | linear interpolation in between  *
	VIS2MM.tCtr_Cust1_In.Y_min_cust		:= -1.0;						* optional: "customized" Y-MIN at the current moment (The existing Y-MIN parameter is the global minimum. To have an effect Y_min_cust needs TO be > the parameter | -1.0 = FUNCTION NOT used *
	VIS2MM.tCtr_Cust1_In.Y_max_cust		:= 1.0;							* optional: "customized" Y-MAX at the current moment (The existing Y-MAX parameter is the global maximum. To have an effect Y_max_cust needs TO be < the parameter | 1.0 = FUNCTION NOT used *
	VIS2MM.tCtr_Cust1_In.Retrigger		:= FALSE;						* optional: a rising EDGE on this input signals the controller to retrigger - set W on X and force the integrator to the current Y  *
	VIS2MM.tCtr_Cust1_In.A;												* optional: feed forward Input *
		xGeACtr_1();	 *FUNCTION call*
	rReplaceMeWithVarname		:= 	OUT_CU.tCtr_Cust1_Out.Y;			*connect actuator variable here*
	OUT_CU.tCtr_CustOut[1].Ao	:= 	OUT_CU.tCtr_Cust1_Out.Y;			*optional: direct hardware output connection with OUT_CU.tCtr_CustOut[x].Ao*
	bReplaceMeWithVarname		:= 	OUT_CU.tCtr_Cust1_Out.Step_down;	*optional: connect actuator variable here for step controller mode*
	bReplaceMeWithVarname		:= 	OUT_CU.tCtr_Cust1_Out.Step_up;		*optional: connect actuator variable here for step controller mode*

	OUT_CU.tCtr_Cust1_In		:= 	VIS2MM.tCtr_Cust1_In;				*forward controller inputs for possible use in other modules*
	OUT_CU.tCtr_Cust1_Out		:= 	MM2VIS.tCtr_Cust1_Out;				*forward controller outputs for possible use in other modules*
	Para.tCtr_Cust1;  													*stated here for watch only*

	******************************************************************************************************************************)

	(* customizable controller 1*)
	VIS2MM.tCtr_Cust1_In.enable			:= Para.bCtr_Cust1 AND TRUE;
	VIS2MM.tCtr_Cust1_In.X				:= 0;
	VIS2MM.tCtr_Cust1_In.W_ext			:= 0;
	VIS2MM.tCtr_Cust1_In.W_ext_Active	:= FALSE;

	VIS2MM.tCtr_Cust1_In.W_set2_Active	:= FALSE;
	VIS2MM.tCtr_Cust1_In.GainScheduling	:= 0.0;
	VIS2MM.tCtr_Cust1_In.Y_min_cust		:= -1.0;
	VIS2MM.tCtr_Cust1_In.Y_max_cust		:= 1.0;
	VIS2MM.tCtr_Cust1_In.Retrigger		:= FALSE;
	VIS2MM.tCtr_Cust1_In.A;

	xGeACtr_1();	(*function call*)
	rReplaceMeWithVarname		:= 	OUT_CU.tCtr_Cust1_Out.Y;
	OUT_CU.tCtr_CustOut[1].Ao	:= 	OUT_CU.tCtr_Cust1_Out.Y;
	bReplaceMeWithVarname		:= 	OUT_CU.tCtr_Cust1_Out.Step_down;
	bReplaceMeWithVarname		:= 	OUT_CU.tCtr_Cust1_Out.Step_up;

	OUT_CU.tCtr_Cust1_In		:= 	VIS2MM.tCtr_Cust1_In;
	OUT_CU.tCtr_Cust1_Out		:= 	MM2VIS.tCtr_Cust1_Out;
	Para.tCtr_Cust1;

	(*******************************************************************************************************************************)
	(* customizable controller 2*)
	VIS2MM.tCtr_Cust2_In.enable			:= Para.bCtr_Cust2 AND TRUE;
	VIS2MM.tCtr_Cust2_In.X				:= 0;
	VIS2MM.tCtr_Cust2_In.W_ext			:= 0;
	VIS2MM.tCtr_Cust2_In.W_ext_Active	:= FALSE;
	VIS2MM.tCtr_Cust2_In.W_set2_Active	:= FALSE;
	VIS2MM.tCtr_Cust2_In.GainScheduling	:= 0.0;
	VIS2MM.tCtr_Cust2_In.Y_min_cust		:= -1.0;
	VIS2MM.tCtr_Cust2_In.Y_max_cust		:= 1.0;
	VIS2MM.tCtr_Cust2_In.Retrigger		:= FALSE;
	VIS2MM.tCtr_Cust2_In.A;

	xGeACtr_2;	(*function call*)
	rReplaceMeWithVarname		:= 	OUT_CU.tCtr_Cust2_Out.Y;
	bReplaceMeWithVarname		:= 	OUT_CU.tCtr_Cust2_Out.Step_down;
	bReplaceMeWithVarname		:= 	OUT_CU.tCtr_Cust2_Out.Step_up;

	OUT_CU.tCtr_Cust2_In		:= 	VIS2MM.tCtr_Cust2_In;
	OUT_CU.tCtr_Cust2_Out		:= 	MM2VIS.tCtr_Cust2_Out;
	Para.tCtr_Cust2;

	(* OPTION to use CtrCust2 as boost temperature controller with humidity function JAPAN Option *)
	OUT_CU.bUseCtrCust2_4HumidityCtr	:= FALSE; (* <-- insert TRUE to use this option *)
	OUT_CU.rCtr_Cust2_W_set				:= Para.tCtr_Cust2.W_set;
	(*******************************************************************************************************************************)
	(* customizable controller 3*)
	VIS2MM.tCtr_Cust3_In.enable			:= Para.bCtr_Cust3 AND TRUE;
	VIS2MM.tCtr_Cust3_In.X				:= 0;
	VIS2MM.tCtr_Cust3_In.W_ext			:= 0;
	VIS2MM.tCtr_Cust3_In.W_ext_Active	:= FALSE;
	VIS2MM.tCtr_Cust3_In.W_set2_Active	:= FALSE;
	VIS2MM.tCtr_Cust3_In.GainScheduling	:= 0.0;
	VIS2MM.tCtr_Cust3_In.Y_min_cust		:= -1.0;
	VIS2MM.tCtr_Cust3_In.Y_max_cust		:= 1.0;
	VIS2MM.tCtr_Cust3_In.Retrigger		:= FALSE;
	VIS2MM.tCtr_Cust3_In.A;

	xGeACtr_3;	(*function call*)
	rReplaceMeWithVarname		:= 	OUT_CU.tCtr_Cust3_Out.Y;
	bReplaceMeWithVarname		:= 	OUT_CU.tCtr_Cust3_Out.Step_down;
	bReplaceMeWithVarname		:= 	OUT_CU.tCtr_Cust3_Out.Step_up;

	OUT_CU.tCtr_Cust3_In		:= 	VIS2MM.tCtr_Cust3_In;
	OUT_CU.tCtr_Cust3_Out		:= 	MM2VIS.tCtr_Cust3_Out;
	Para.tCtr_Cust3;

	(*******************************************************************************************************************************)
	(* customizable controller 4*)
	VIS2MM.tCtr_Cust4_In.enable			:= Para.bCtr_Cust4 AND TRUE;
	VIS2MM.tCtr_Cust4_In.X				:= 0;
	VIS2MM.tCtr_Cust4_In.W_ext			:= 0;
	VIS2MM.tCtr_Cust4_In.W_ext_Active	:= FALSE;
	VIS2MM.tCtr_Cust4_In.W_set2_Active	:= FALSE;
	VIS2MM.tCtr_Cust4_In.GainScheduling	:= 0.0;
	VIS2MM.tCtr_Cust4_In.Y_min_cust		:= -1.0;
	VIS2MM.tCtr_Cust4_In.Y_max_cust		:= 1.0;
	VIS2MM.tCtr_Cust4_In.Retrigger		:= FALSE;
	VIS2MM.tCtr_Cust4_In.A;

	xGeACtr_4;	(*function call*)
	rReplaceMeWithVarname		:= 	OUT_CU.tCtr_Cust4_Out.Y;
	bReplaceMeWithVarname		:= 	OUT_CU.tCtr_Cust4_Out.Step_down;
	bReplaceMeWithVarname		:= 	OUT_CU.tCtr_Cust4_Out.Step_up;

	OUT_CU.tCtr_Cust4_In		:= 	VIS2MM.tCtr_Cust4_In;
	OUT_CU.tCtr_Cust4_Out		:= 	MM2VIS.tCtr_Cust4_Out;
	Para.tCtr_Cust4;

	(*******************************************************************************************************************************)
	(* customizable controller 5*)
	VIS2MM.tCtr_Cust5_In.enable			:= Para.bCtr_Cust5 AND TRUE;
	VIS2MM.tCtr_Cust5_In.X				:= 0;
	VIS2MM.tCtr_Cust5_In.W_ext			:= 0;
	VIS2MM.tCtr_Cust5_In.W_ext_Active	:= FALSE;
	VIS2MM.tCtr_Cust5_In.W_set2_Active	:= FALSE;
	VIS2MM.tCtr_Cust5_In.GainScheduling	:= 0.0;
	VIS2MM.tCtr_Cust5_In.Y_min_cust		:= -1.0;
	VIS2MM.tCtr_Cust5_In.Y_max_cust		:= 1.0;
	VIS2MM.tCtr_Cust5_In.Retrigger		:= FALSE;
	VIS2MM.tCtr_Cust5_In.A;

	xGeACtr_5;	(*function call*)
	rReplaceMeWithVarname		:= 	OUT_CU.tCtr_Cust5_Out.Y;
	bReplaceMeWithVarname		:= 	OUT_CU.tCtr_Cust5_Out.Step_down;
	bReplaceMeWithVarname		:= 	OUT_CU.tCtr_Cust5_Out.Step_up;

	OUT_CU.tCtr_Cust5_In		:= 	VIS2MM.tCtr_Cust5_In;
	OUT_CU.tCtr_Cust5_Out		:= 	MM2VIS.tCtr_Cust5_Out;
	Para.tCtr_Cust5;

	(*******************************************************************************************************************************)
	(* customizable controller 6*)
	VIS2MM.tCtr_Cust6_In.enable			:= Para.bCtr_Cust6 AND TRUE;
	VIS2MM.tCtr_Cust6_In.X				:= 0;
	VIS2MM.tCtr_Cust6_In.W_ext			:= 0;
	VIS2MM.tCtr_Cust6_In.W_ext_Active	:= FALSE;
	VIS2MM.tCtr_Cust6_In.W_set2_Active	:= FALSE;
	VIS2MM.tCtr_Cust6_In.GainScheduling	:= 0.0;
	VIS2MM.tCtr_Cust6_In.Y_min_cust		:= -1.0;
	VIS2MM.tCtr_Cust6_In.Y_max_cust		:= 1.0;
	VIS2MM.tCtr_Cust6_In.Retrigger		:= FALSE;
	VIS2MM.tCtr_Cust6_In.A;

	xGeACtr_6;	(*function call*)
	rReplaceMeWithVarname		:= 	OUT_CU.tCtr_Cust6_Out.Y;
	bReplaceMeWithVarname		:= 	OUT_CU.tCtr_Cust6_Out.Step_down;
	bReplaceMeWithVarname		:= 	OUT_CU.tCtr_Cust6_Out.Step_up;

	OUT_CU.tCtr_Cust6_In		:= 	VIS2MM.tCtr_Cust6_In;
	OUT_CU.tCtr_Cust6_Out		:= 	MM2VIS.tCtr_Cust6_Out;
	Para.tCtr_Cust6;

	(*******************************************************************************************************************************)
	(* customizable controller 7*)
	VIS2MM.tCtr_Cust7_In.enable			:= Para.bCtr_Cust7 AND TRUE;
	VIS2MM.tCtr_Cust7_In.X				:= 0;
	VIS2MM.tCtr_Cust7_In.W_ext			:= 0;
	VIS2MM.tCtr_Cust7_In.W_ext_Active	:= FALSE;
	VIS2MM.tCtr_Cust7_In.W_set2_Active	:= FALSE;
	VIS2MM.tCtr_Cust7_In.GainScheduling	:= 0.0;
	VIS2MM.tCtr_Cust7_In.Y_min_cust		:= -1.0;
	VIS2MM.tCtr_Cust7_In.Y_max_cust		:= 1.0;
	VIS2MM.tCtr_Cust7_In.Retrigger		:= FALSE;
	VIS2MM.tCtr_Cust7_In.A;

	xGeACtr_7;	(*function call*)
	rReplaceMeWithVarname		:= 	OUT_CU.tCtr_Cust7_Out.Y;
	bReplaceMeWithVarname		:= 	OUT_CU.tCtr_Cust7_Out.Step_down;
	bReplaceMeWithVarname		:= 	OUT_CU.tCtr_Cust7_Out.Step_up;

	OUT_CU.tCtr_Cust7_In		:= 	VIS2MM.tCtr_Cust7_In;
	OUT_CU.tCtr_Cust7_Out		:= 	MM2VIS.tCtr_Cust7_Out;
	Para.tCtr_Cust7;

	(*******************************************************************************************************************************)
	(* customizable controller 8*)
	VIS2MM.tCtr_Cust8_In.enable			:= Para.bCtr_Cust8 AND TRUE;
	VIS2MM.tCtr_Cust8_In.X				:= 0;
	VIS2MM.tCtr_Cust8_In.W_ext			:= 0;
	VIS2MM.tCtr_Cust8_In.W_ext_Active	:= FALSE;
	VIS2MM.tCtr_Cust8_In.W_set2_Active	:= FALSE;
	VIS2MM.tCtr_Cust8_In.GainScheduling	:= 0.0;
	VIS2MM.tCtr_Cust8_In.Y_min_cust		:= -1.0;
	VIS2MM.tCtr_Cust8_In.Y_max_cust		:= 1.0;
	VIS2MM.tCtr_Cust8_In.Retrigger		:= FALSE;
	VIS2MM.tCtr_Cust8_In.A;

	xGeACtr_8;	(*function call*)
	rReplaceMeWithVarname		:= 	OUT_CU.tCtr_Cust8_Out.Y;
	bReplaceMeWithVarname		:= 	OUT_CU.tCtr_Cust8_Out.Step_down;
	bReplaceMeWithVarname		:= 	OUT_CU.tCtr_Cust8_Out.Step_up;

	OUT_CU.tCtr_Cust8_In		:= 	VIS2MM.tCtr_Cust8_In;
	OUT_CU.tCtr_Cust8_Out		:= 	MM2VIS.tCtr_Cust8_Out;
	Para.tCtr_Cust8;

	(*******************************************************************************************************************************)
	(* customizable controller 41*)		(* extended controller items 41-45 ONLY FOR USE WITH HMI Extension Package!*)
	VIS2MM.tCtr_Cust41_In.enable		:= Para.bCtr_Cust41 AND TRUE;
	VIS2MM.tCtr_Cust41_In.X				:= 0;
	VIS2MM.tCtr_Cust41_In.W_ext			:= 0;
	VIS2MM.tCtr_Cust41_In.W_ext_Active	:= FALSE;
	VIS2MM.tCtr_Cust41_In.W_set2_Active	:= FALSE;
	VIS2MM.tCtr_Cust41_In.GainScheduling:= 0.0;
	VIS2MM.tCtr_Cust41_In.Y_min_cust	:= -1.0;
	VIS2MM.tCtr_Cust41_In.Y_max_cust	:= 1.0;
	VIS2MM.tCtr_Cust41_In.Retrigger		:= FALSE;
	VIS2MM.tCtr_Cust41_In.A;

	xGeACtr_41;	(*function call*)
	rReplaceMeWithVarname		:= 	OUT_CU.tCtr_Cust41_Out.Y;
	bReplaceMeWithVarname		:= 	OUT_CU.tCtr_Cust41_Out.Step_down;
	bReplaceMeWithVarname		:= 	OUT_CU.tCtr_Cust41_Out.Step_up;

	OUT_CU.tCtr_Cust41_In		:= 	VIS2MM.tCtr_Cust41_In;
	OUT_CU.tCtr_Cust41_Out		:= 	MM2VIS.tCtr_Cust41_Out;
	Para.tCtr_Cust41;

	(*******************************************************************************************************************************)
	(* customizable controller 42*)
	VIS2MM.tCtr_Cust42_In.enable		:= Para.bCtr_Cust42 AND TRUE;
	VIS2MM.tCtr_Cust42_In.X				:= 0;
	VIS2MM.tCtr_Cust42_In.W_ext			:= 0;
	VIS2MM.tCtr_Cust42_In.W_ext_Active	:= FALSE;
	VIS2MM.tCtr_Cust42_In.W_set2_Active	:= FALSE;
	VIS2MM.tCtr_Cust42_In.GainScheduling:= 0.0;
	VIS2MM.tCtr_Cust42_In.Y_min_cust	:= -1.0;
	VIS2MM.tCtr_Cust42_In.Y_max_cust	:= 1.0;
	VIS2MM.tCtr_Cust42_In.Retrigger		:= FALSE;
	VIS2MM.tCtr_Cust42_In.A;

	xGeACtr_42;	(*function call*)
	rReplaceMeWithVarname		:= 	OUT_CU.tCtr_Cust42_Out.Y;
	bReplaceMeWithVarname		:= 	OUT_CU.tCtr_Cust42_Out.Step_down;
	bReplaceMeWithVarname		:= 	OUT_CU.tCtr_Cust42_Out.Step_up;

	OUT_CU.tCtr_Cust42_In		:= 	VIS2MM.tCtr_Cust42_In;
	OUT_CU.tCtr_Cust42_Out		:= 	MM2VIS.tCtr_Cust42_Out;
	Para.tCtr_Cust42;

	(*******************************************************************************************************************************)
	(* customizable controller 43*)
	VIS2MM.tCtr_Cust43_In.enable		:= Para.bCtr_Cust43 AND TRUE;
	VIS2MM.tCtr_Cust43_In.X				:= 0;
	VIS2MM.tCtr_Cust43_In.W_ext			:= 0;
	VIS2MM.tCtr_Cust43_In.W_ext_Active	:= FALSE;
	VIS2MM.tCtr_Cust43_In.W_set2_Active	:= FALSE;
	VIS2MM.tCtr_Cust43_In.GainScheduling:= 0.0;
	VIS2MM.tCtr_Cust43_In.Y_min_cust	:= -1.0;
	VIS2MM.tCtr_Cust43_In.Y_max_cust	:= 1.0;
	VIS2MM.tCtr_Cust43_In.Retrigger		:= FALSE;
	VIS2MM.tCtr_Cust43_In.A;

	xGeACtr_43;	(*function call*)
	rReplaceMeWithVarname		:= 	OUT_CU.tCtr_Cust43_Out.Y;
	bReplaceMeWithVarname		:= 	OUT_CU.tCtr_Cust43_Out.Step_down;
	bReplaceMeWithVarname		:= 	OUT_CU.tCtr_Cust43_Out.Step_up;

	OUT_CU.tCtr_Cust43_In		:= 	VIS2MM.tCtr_Cust43_In;
	OUT_CU.tCtr_Cust43_Out		:= 	MM2VIS.tCtr_Cust43_Out;
	Para.tCtr_Cust43;

	(*******************************************************************************************************************************)
	(* customizable controller 44*)
	VIS2MM.tCtr_Cust44_In.enable		:= Para.bCtr_Cust44 AND TRUE;
	VIS2MM.tCtr_Cust44_In.X				:= 0;
	VIS2MM.tCtr_Cust44_In.W_ext			:= 0;
	VIS2MM.tCtr_Cust44_In.W_ext_Active	:= FALSE;
	VIS2MM.tCtr_Cust44_In.W_set2_Active	:= FALSE;
	VIS2MM.tCtr_Cust44_In.GainScheduling:= 0.0;
	VIS2MM.tCtr_Cust44_In.Y_min_cust	:= -1.0;
	VIS2MM.tCtr_Cust44_In.Y_max_cust	:= 1.0;
	VIS2MM.tCtr_Cust44_In.Retrigger		:= FALSE;
	VIS2MM.tCtr_Cust44_In.A;

	xGeACtr_44;	(*function call*)
	rReplaceMeWithVarname		:= 	OUT_CU.tCtr_Cust44_Out.Y;
	bReplaceMeWithVarname		:= 	OUT_CU.tCtr_Cust44_Out.Step_down;
	bReplaceMeWithVarname		:= 	OUT_CU.tCtr_Cust44_Out.Step_up;

	OUT_CU.tCtr_Cust44_In		:= 	VIS2MM.tCtr_Cust44_In;
	OUT_CU.tCtr_Cust44_Out		:= 	MM2VIS.tCtr_Cust44_Out;
	Para.tCtr_Cust44;

	(*******************************************************************************************************************************)
	(* customizable controller 45*)
	VIS2MM.tCtr_Cust45_In.enable		:= Para.bCtr_Cust45 AND TRUE;
	VIS2MM.tCtr_Cust45_In.X				:= 0;
	VIS2MM.tCtr_Cust45_In.W_ext			:= 0;
	VIS2MM.tCtr_Cust45_In.W_ext_Active	:= FALSE;
	VIS2MM.tCtr_Cust45_In.W_set2_Active	:= FALSE;
	VIS2MM.tCtr_Cust45_In.GainScheduling:= 0.0;
	VIS2MM.tCtr_Cust45_In.Y_min_cust	:= -1.0;
	VIS2MM.tCtr_Cust45_In.Y_max_cust	:= 1.0;
	VIS2MM.tCtr_Cust45_In.A;

	xGeACtr_45;	(*function call*)
	rReplaceMeWithVarname		:= 	OUT_CU.tCtr_Cust45_Out.Y;
	bReplaceMeWithVarname		:= 	OUT_CU.tCtr_Cust45_Out.Step_down;
	bReplaceMeWithVarname		:= 	OUT_CU.tCtr_Cust45_Out.Step_up;

	OUT_CU.tCtr_Cust45_In		:= 	VIS2MM.tCtr_Cust45_In;
	OUT_CU.tCtr_Cust45_Out		:= 	MM2VIS.tCtr_Cust45_Out;
	Para.tCtr_Cust45;

END_PROGRAM
```

#### c_ctrInit.st - Initialization code
```iecst
(*******************************************************************************
CUSTOMIZED: c_ctr 		reserve controller handling (init)

This code is confidential AND proprietary to the INNIO Company.
It may NOT be used in any form, or reproduced in any manner,
without written permission of the INNIO Company.
Copyright, INNIO Company, 2022

Customized modifications: -
------------------------

History:
-------
		23.05.2012	Zengerer	generated, new
V4.02	09.09.2015	Zengerer	cleanup, prototype entry FOR documentation comments
V4.04	20.06.2016	Weitzer		add controller 41 .. 45
V4.11	27.01.2022	Perktold	impemented plant controller upgrade (AlwaysUseYRamp, KeepYManAtBlock both signals Std. TRUE)

Instructions for use:
--------------------
-
Outstandings:
------------
-

*******************************************************************************)

PROGRAM _INIT

	(*Parameter FACTORY DEFAULT VALUES *)
	(*for missing/new/not visualized parameter*)
	ParaFactoryDefault.tCtr_Cust1.t_min_pulse_down :=	10;
	ParaFactoryDefault.tCtr_Cust1.t_min_pulse_up :=		10;
	ParaFactoryDefault.tCtr_Cust1.t_period_down :=		100;
	ParaFactoryDefault.tCtr_Cust1.t_period_up :=		100;

	(*REG2*)
	ParaFactoryDefault.tCtr_Cust2.t_min_pulse_down :=	10;
	ParaFactoryDefault.tCtr_Cust2.t_min_pulse_up :=		10;
	ParaFactoryDefault.tCtr_Cust2.t_period_down :=		100;
	ParaFactoryDefault.tCtr_Cust2.t_period_up :=		100;

	(*REG3*)
	ParaFactoryDefault.tCtr_Cust3.t_min_pulse_down :=	10;
	ParaFactoryDefault.tCtr_Cust3.t_min_pulse_up :=		10;
	ParaFactoryDefault.tCtr_Cust3.t_period_down :=		100;
	ParaFactoryDefault.tCtr_Cust3.t_period_up :=		100;

	(*REG4*)
	ParaFactoryDefault.tCtr_Cust4.t_min_pulse_down :=	10;
	ParaFactoryDefault.tCtr_Cust4.t_min_pulse_up :=		10;
	ParaFactoryDefault.tCtr_Cust4.t_period_down :=		100;
	ParaFactoryDefault.tCtr_Cust4.t_period_up :=		100;

	(*REG5*)
	ParaFactoryDefault.tCtr_Cust5.t_min_pulse_down :=	10;
	ParaFactoryDefault.tCtr_Cust5.t_min_pulse_up :=		10;
	ParaFactoryDefault.tCtr_Cust5.t_period_down :=		100;
	ParaFactoryDefault.tCtr_Cust5.t_period_up :=		100;

	(*REG6*)
	ParaFactoryDefault.tCtr_Cust6.t_min_pulse_down :=	10;
	ParaFactoryDefault.tCtr_Cust6.t_min_pulse_up :=		10;
	ParaFactoryDefault.tCtr_Cust6.t_period_down :=		100;
	ParaFactoryDefault.tCtr_Cust6.t_period_up :=		100;

	(*REG7*)
	ParaFactoryDefault.tCtr_Cust7.t_min_pulse_down :=	10;
	ParaFactoryDefault.tCtr_Cust7.t_min_pulse_up :=		10;
	ParaFactoryDefault.tCtr_Cust7.t_period_down :=		100;
	ParaFactoryDefault.tCtr_Cust7.t_period_up :=		100;

	(*REG8*)
	ParaFactoryDefault.tCtr_Cust8.t_min_pulse_down :=	10;
	ParaFactoryDefault.tCtr_Cust8.t_min_pulse_up :=		10;
	ParaFactoryDefault.tCtr_Cust8.t_period_down :=		100;
	ParaFactoryDefault.tCtr_Cust8.t_period_up :=		100;

	(*REG41*)
	ParaFactoryDefault.tCtr_Cust41.t_min_pulse_down :=	10;
	ParaFactoryDefault.tCtr_Cust41.t_min_pulse_up :=	10;
	ParaFactoryDefault.tCtr_Cust41.t_period_down :=		100;
	ParaFactoryDefault.tCtr_Cust41.t_period_up :=		100;

	(*REG42*)
	ParaFactoryDefault.tCtr_Cust42.t_min_pulse_down :=	10;
	ParaFactoryDefault.tCtr_Cust42.t_min_pulse_up :=	10;
	ParaFactoryDefault.tCtr_Cust42.t_period_down :=		100;
	ParaFactoryDefault.tCtr_Cust42.t_period_up :=		100;

	(*REG43*)
	ParaFactoryDefault.tCtr_Cust43.t_min_pulse_down :=	10;
	ParaFactoryDefault.tCtr_Cust43.t_min_pulse_up :=	10;
	ParaFactoryDefault.tCtr_Cust43.t_period_down :=		100;
	ParaFactoryDefault.tCtr_Cust43.t_period_up :=		100;

	(*REG44*)
	ParaFactoryDefault.tCtr_Cust44.t_min_pulse_down :=	10;
	ParaFactoryDefault.tCtr_Cust44.t_min_pulse_up :=	10;
	ParaFactoryDefault.tCtr_Cust44.t_period_down :=		100;
	ParaFactoryDefault.tCtr_Cust44.t_period_up :=		100;

	(*REG45*)
	ParaFactoryDefault.tCtr_Cust45.t_min_pulse_down :=	10;
	ParaFactoryDefault.tCtr_Cust45.t_min_pulse_up :=	10;
	ParaFactoryDefault.tCtr_Cust45.t_period_down :=		100;
	ParaFactoryDefault.tCtr_Cust45.t_period_up :=		100;

	(*avoid status 12033 error*)
	IF Para.tCtr_Cust1.t_period_up = 0 		THEN Para.tCtr_Cust1.t_period_up := 100; 	END_IF	(*avoid status 12033 error*)
	IF Para.tCtr_Cust1.t_period_down = 0 	THEN Para.tCtr_Cust1.t_period_down := 100; 	END_IF
	IF Para.tCtr_Cust2.t_period_up = 0 		THEN Para.tCtr_Cust2.t_period_up := 100; 	END_IF
	IF Para.tCtr_Cust2.t_period_down = 0 	THEN Para.tCtr_Cust2.t_period_down := 100; 	END_IF
	IF Para.tCtr_Cust3.t_period_up = 0 		THEN Para.tCtr_Cust3.t_period_up := 100; 	END_IF
	IF Para.tCtr_Cust3.t_period_down = 0 	THEN Para.tCtr_Cust3.t_period_down := 100; 	END_IF
	IF Para.tCtr_Cust4.t_period_up = 0 		THEN Para.tCtr_Cust4.t_period_up := 100; 	END_IF
	IF Para.tCtr_Cust4.t_period_down = 0 	THEN Para.tCtr_Cust4.t_period_down := 100; 	END_IF
	IF Para.tCtr_Cust5.t_period_up = 0 		THEN Para.tCtr_Cust5.t_period_up := 100; 	END_IF
	IF Para.tCtr_Cust5.t_period_down = 0 	THEN Para.tCtr_Cust5.t_period_down := 100; 	END_IF
	IF Para.tCtr_Cust6.t_period_up = 0 		THEN Para.tCtr_Cust6.t_period_up := 100; 	END_IF
	IF Para.tCtr_Cust6.t_period_down = 0 	THEN Para.tCtr_Cust6.t_period_down := 100; 	END_IF
	IF Para.tCtr_Cust7.t_period_up = 0 		THEN Para.tCtr_Cust7.t_period_up := 100; 	END_IF
	IF Para.tCtr_Cust7.t_period_down = 0 	THEN Para.tCtr_Cust7.t_period_down := 100; 	END_IF
	IF Para.tCtr_Cust8.t_period_up = 0 		THEN Para.tCtr_Cust8.t_period_up := 100; 	END_IF
	IF Para.tCtr_Cust8.t_period_down = 0 	THEN Para.tCtr_Cust8.t_period_down := 100; 	END_IF

	IF Para.tCtr_Cust41.t_period_up = 0 	THEN Para.tCtr_Cust41.t_period_up := 100; 	END_IF
	IF Para.tCtr_Cust41.t_period_down = 0 	THEN Para.tCtr_Cust41.t_period_down := 100;	END_IF
	IF Para.tCtr_Cust42.t_period_up = 0 	THEN Para.tCtr_Cust42.t_period_up := 100; 	END_IF
	IF Para.tCtr_Cust42.t_period_down = 0 	THEN Para.tCtr_Cust42.t_period_down := 100; END_IF
	IF Para.tCtr_Cust43.t_period_up = 0 	THEN Para.tCtr_Cust43.t_period_up := 100; 	END_IF
	IF Para.tCtr_Cust43.t_period_down = 0 	THEN Para.tCtr_Cust43.t_period_down := 100; END_IF
	IF Para.tCtr_Cust44.t_period_up = 0 	THEN Para.tCtr_Cust44.t_period_up := 100; 	END_IF
	IF Para.tCtr_Cust44.t_period_down = 0 	THEN Para.tCtr_Cust44.t_period_down := 100; END_IF
	IF Para.tCtr_Cust45.t_period_up = 0 	THEN Para.tCtr_Cust45.t_period_up := 100; 	END_IF
	IF Para.tCtr_Cust45.t_period_down = 0 	THEN Para.tCtr_Cust45.t_period_down := 100; END_IF

	VIS2MM.tCtr_Cust1_In.AlwaysUseYRamp		:= TRUE;	(*If TRUE the Y signal will always limit the change rate via the according parameter | if FALSE the Y signal will jump in case the controller is disabled (blocked or set)*)
	VIS2MM.tCtr_Cust1_In.KeepYManAtBlock	:= TRUE;	(*If TRUE the controller will keep the Y-man value constant in case the controller is disabled (blocked or set) | If FALSE the blocked or set value will override the Y-man value*)
	VIS2MM.tCtr_Cust1_In.Y_min_cust			:= -1.0;	(*"customized" Y-Min at the current moment (The existing Y-Min parameter is the global minimum. To have an effect Y_min_cust needs to be > the parameter | -1.0 = function not used*)
	VIS2MM.tCtr_Cust1_In.Y_max_cust			:=  1.0;	(*"customized" Y-Max at the current moment (The existing Y-Max parameter is the global maximum. To have an effect Y_max_cust needs to be < the parameter | 1.0 = function not used*)
	VIS2MM.tCtr_Cust1_In.StepperMode		:= FALSE;	(* TRUE = use PWM-Mode (standard mode until 4.10) | FALSE = use continuous servo drive *)
	VIS2MM.tCtr_Cust2_In.AlwaysUseYRamp		:= TRUE;
	VIS2MM.tCtr_Cust2_In.KeepYManAtBlock	:= TRUE;
	VIS2MM.tCtr_Cust2_In.Y_min_cust			:= -1.0;
	VIS2MM.tCtr_Cust2_In.Y_max_cust			:=  1.0;
	VIS2MM.tCtr_Cust2_In.StepperMode		:= FALSE;
	VIS2MM.tCtr_Cust3_In.AlwaysUseYRamp		:= TRUE;
	VIS2MM.tCtr_Cust3_In.KeepYManAtBlock	:= TRUE;
	VIS2MM.tCtr_Cust3_In.Y_min_cust			:= -1.0;
	VIS2MM.tCtr_Cust3_In.Y_max_cust			:=  1.0;
	VIS2MM.tCtr_Cust3_In.StepperMode		:= FALSE;
	VIS2MM.tCtr_Cust4_In.AlwaysUseYRamp		:= TRUE;
	VIS2MM.tCtr_Cust4_In.KeepYManAtBlock	:= TRUE;
	VIS2MM.tCtr_Cust4_In.Y_min_cust			:= -1.0;
	VIS2MM.tCtr_Cust4_In.Y_max_cust			:=  1.0;
	VIS2MM.tCtr_Cust4_In.StepperMode		:= FALSE;

	VIS2MM.tCtr_Cust5_In.AlwaysUseYRamp		:= TRUE;
	VIS2MM.tCtr_Cust5_In.KeepYManAtBlock	:= TRUE;
	VIS2MM.tCtr_Cust5_In.Y_min_cust			:= -1.0;
	VIS2MM.tCtr_Cust5_In.Y_max_cust			:=  1.0;
	VIS2MM.tCtr_Cust5_In.StepperMode		:= FALSE;
	VIS2MM.tCtr_Cust6_In.AlwaysUseYRamp		:= TRUE;
	VIS2MM.tCtr_Cust6_In.KeepYManAtBlock	:= TRUE;
	VIS2MM.tCtr_Cust6_In.Y_min_cust			:= -1.0;
	VIS2MM.tCtr_Cust6_In.Y_max_cust			:=  1.0;
	VIS2MM.tCtr_Cust6_In.StepperMode		:= FALSE;
	VIS2MM.tCtr_Cust7_In.AlwaysUseYRamp		:= TRUE;
	VIS2MM.tCtr_Cust7_In.KeepYManAtBlock	:= TRUE;
	VIS2MM.tCtr_Cust7_In.Y_min_cust			:= -1.0;
	VIS2MM.tCtr_Cust7_In.Y_max_cust			:=  1.0;
	VIS2MM.tCtr_Cust7_In.StepperMode		:= FALSE;
	VIS2MM.tCtr_Cust8_In.AlwaysUseYRamp		:= TRUE;
	VIS2MM.tCtr_Cust8_In.KeepYManAtBlock	:= TRUE;
	VIS2MM.tCtr_Cust8_In.Y_min_cust			:= -1.0;
	VIS2MM.tCtr_Cust8_In.Y_max_cust			:=  1.0;
	VIS2MM.tCtr_Cust8_In.StepperMode		:= FALSE;

	VIS2MM.tCtr_Cust41_In.AlwaysUseYRamp	:= TRUE;
	VIS2MM.tCtr_Cust41_In.KeepYManAtBlock	:= TRUE;
	VIS2MM.tCtr_Cust41_In.Y_min_cust		:= -1.0;
	VIS2MM.tCtr_Cust41_In.Y_max_cust		:=  1.0;
	VIS2MM.tCtr_Cust41_In.StepperMode		:= FALSE;
	VIS2MM.tCtr_Cust42_In.AlwaysUseYRamp	:= TRUE;
	VIS2MM.tCtr_Cust42_In.KeepYManAtBlock	:= TRUE;
	VIS2MM.tCtr_Cust42_In.Y_min_cust		:= -1.0;
	VIS2MM.tCtr_Cust42_In.Y_max_cust		:=  1.0;
	VIS2MM.tCtr_Cust42_In.StepperMode		:= FALSE;
	VIS2MM.tCtr_Cust43_In.AlwaysUseYRamp	:= TRUE;
	VIS2MM.tCtr_Cust43_In.KeepYManAtBlock	:= TRUE;
	VIS2MM.tCtr_Cust43_In.Y_min_cust		:= -1.0;
	VIS2MM.tCtr_Cust43_In.Y_max_cust		:=  1.0;
	VIS2MM.tCtr_Cust43_In.StepperMode		:= FALSE;
	VIS2MM.tCtr_Cust44_In.AlwaysUseYRamp	:= TRUE;
	VIS2MM.tCtr_Cust44_In.KeepYManAtBlock	:= TRUE;
	VIS2MM.tCtr_Cust44_In.Y_min_cust		:= -1.0;
	VIS2MM.tCtr_Cust44_In.Y_max_cust		:=  1.0;
	VIS2MM.tCtr_Cust44_In.StepperMode		:= FALSE;

(* configure and asign structures for customizable controllers *)

	(* configure and asign structures for customizable controllers *)
	xGeACtr_1(pParameter := ADR(Para.tCtr_Cust1), pInput := ADR(VIS2MM.tCtr_Cust1_In), pOutput := ADR(MM2VIS.tCtr_Cust1_Out));
	xGeACtr_2(pParameter := ADR(Para.tCtr_Cust2), pInput := ADR(VIS2MM.tCtr_Cust2_In), pOutput := ADR(MM2VIS.tCtr_Cust2_Out));
	xGeACtr_3(pParameter := ADR(Para.tCtr_Cust3), pInput := ADR(VIS2MM.tCtr_Cust3_In), pOutput := ADR(MM2VIS.tCtr_Cust3_Out));
	xGeACtr_4(pParameter := ADR(Para.tCtr_Cust4), pInput := ADR(VIS2MM.tCtr_Cust4_In), pOutput := ADR(MM2VIS.tCtr_Cust4_Out));

	xGeACtr_5(pParameter := ADR(Para.tCtr_Cust5), pInput := ADR(VIS2MM.tCtr_Cust5_In), pOutput := ADR(MM2VIS.tCtr_Cust5_Out));
	xGeACtr_6(pParameter := ADR(Para.tCtr_Cust6), pInput := ADR(VIS2MM.tCtr_Cust6_In), pOutput := ADR(MM2VIS.tCtr_Cust6_Out));
	xGeACtr_7(pParameter := ADR(Para.tCtr_Cust7), pInput := ADR(VIS2MM.tCtr_Cust7_In), pOutput := ADR(MM2VIS.tCtr_Cust7_Out));
	xGeACtr_8(pParameter := ADR(Para.tCtr_Cust8), pInput := ADR(VIS2MM.tCtr_Cust8_In), pOutput := ADR(MM2VIS.tCtr_Cust8_Out));

	xGeACtr_41(pParameter := ADR(Para.tCtr_Cust41), pInput := ADR(VIS2MM.tCtr_Cust41_In), pOutput := ADR(MM2VIS.tCtr_Cust41_Out));
	xGeACtr_42(pParameter := ADR(Para.tCtr_Cust42), pInput := ADR(VIS2MM.tCtr_Cust42_In), pOutput := ADR(MM2VIS.tCtr_Cust42_Out));
	xGeACtr_43(pParameter := ADR(Para.tCtr_Cust43), pInput := ADR(VIS2MM.tCtr_Cust43_In), pOutput := ADR(MM2VIS.tCtr_Cust43_Out));
	xGeACtr_44(pParameter := ADR(Para.tCtr_Cust44), pInput := ADR(VIS2MM.tCtr_Cust44_In), pOutput := ADR(MM2VIS.tCtr_Cust44_Out));
	xGeACtr_45(pParameter := ADR(Para.tCtr_Cust45), pInput := ADR(VIS2MM.tCtr_Cust45_In), pOutput := ADR(MM2VIS.tCtr_Cust45_Out));

END_PROGRAM
```

#### c_ctr.var - Local variables
```iecst
(********************************************************************
 * COPYRIGHT -- INNIO Company
 ********************************************************************
 * Program: c_ctr
 * File: c_ctr.var
 * Author: ZengereS
 * Created: May 30, 2012
 ********************************************************************
 * Local variables of program c_ctr
 ********************************************************************)
VAR
	xGeACtr_1 : GeACtr;
	xGeACtr_2 : GeACtr;
	xGeACtr_3 : GeACtr;
	xGeACtr_4 : GeACtr;
	xGeACtr_5 : GeACtr;
	xGeACtr_6 : GeACtr;
	xGeACtr_7 : GeACtr;
	xGeACtr_8 : GeACtr;
	xGeACtr_41 : GeACtr;
	xGeACtr_42 : GeACtr;
	xGeACtr_43 : GeACtr;
	xGeACtr_44 : GeACtr;
	xGeACtr_45 : GeACtr;
	rReplaceMeWithVarname : REAL; (*void*)
	bReplaceMeWithVarname : BOOL; (*void*)
END_VAR
```

### Program Logical/Customized/c_cnt (IEC, version 4.10.0) - Counter Task th handle customizable counters

#### counterCyclic.st
```iecst
(*******************************************************************************
AGGR: counter.st - connection and processing of counters (cyclic)

This code is confidential and proprietary to the INNIO Company.
It may not be used in any form, or reproduced in any manner, without the express
written permission of the INNIO Company.
Copyright, INNIO Company, 2016

- preparation of the RPS time (if necessary for compatibility)
- prepare evaluation of the impulses
- evaluation of the maintenance counter
- evaluation reserve counter

Customized modifications:
------------------------

History:
-------
V3.90	05.07.2012 Zengerer	NEW SEPARATED PART for MM_Customized, derived from V3.20	03-11-2010	Weitzer
V3.91	08.08.2012 Zengerer iCnt_OpHours replaces start_z (rCnt_OpHours), iCnt_Starts replaces betrieb_h (rCnt_Starts)
V3.92	07.09.2012 Zengerer bRPM_Count.. replaces RPMZ..
V3.93	12.11.2012 Zengerer	Counter moved to IN_CU.iCount.. to allow user input
V3.94	05.12.2012 Zengerer	expanded to 10 counters
V4.02	07.10.2015 Zengerer	bOpt_100msTakClock to activate msec counter function with iCount10
V4.04	20.06.2016 Weitzer	add reserve counter 11..20
V4.07	11.10.2018 Zengerer task moved  to 10ms TC#2 to handle inputs down to minimum frequency <49Hz
							new IN_CU.tCustDigIn_TC2[1].Di for task input bits in 10ms TC#2 VVM, to handle 5Hz to <=49Hz inputs!
V4.07.03 10.09.2019 Zen		Mind changed Perm Storage Handling for reduced file write cycle in task Perm_CU
V4.10.90BETA .2020 Zengerer	Remove example connection
V4.10 	03.12.2020 Zengerer MaintenanceCount reset interlock to IN_CU.iCnt_Starts
V4.11	17.02.2022 Zengerer extended counter items 11- ONLY FOR USE WITH HMI Extension Package import

Instructions for use:
--------------------
- connect (or replace) bConnectYourBitToCountHere,  according customer needs
- connect IN_CU.bRPM_Count1...IN_CU.bRPM_Count16,  according customer needs in other Modules or
			replace <bConnectYourBitToStartTimeHere> with local variable
- optional set bOpt_10msTaskClock = TRUE TO activate msec counter FUNCTION with iCount20

Outstandings:
------------
V4.07: watch out to copy your task input bit in 10ms TC#2 VVM, to handle 5Hz to <=49Hz inputs!

*********************************************************************************)

PROGRAM _CYCLIC

	(* reserve counter 1 *)
	xImp_Count_1.CLK 	:= bConnectYourBitToCountHere1 ;	// := IN_CU.tCustDigCnt_TC2[1].Di;		(* change customized; !Watch out to copy your task input bit in 10ms TC#2 VVM, to handle >5Hz to <=49Hz inputs! *)
	xImp_Count_1;	(* call FUB R_TRIG *)

	(* reserve counter 2 *)
	xImp_Count_2.CLK 	:= bConnectYourBitToCountHere2; 			(* change customized (old: zaehl_2)  *)
	xImp_Count_2;	(* call FUB R_TRIG *)

	(* reserve counter 3 *)
	xImp_Count_3.CLK 	:= bConnectYourBitToCountHere3;				(* change customized  (old: zaehl_3) *)
	xImp_Count_3;	(* call FUB R_TRIG *)

	(* reserve counter 4 *)
	xImp_Count_4.CLK 	:= bConnectYourBitToCountHere4;  			(* change customized   (old: zaehl_4) *)
	xImp_Count_4;	(* call FUB R_TRIG *)

	(* reserve counter 5 *)
	xImp_Count_5.CLK 	:=  bConnectYourBitToCountHere;					(* change customized *)
	xImp_Count_5;	(* call FUB R_TRIG *)

	(* reserve counter 6 *)
	xImp_Count_6.CLK 	:= bConnectYourBitToCountHere; 					(* change customized *)
	xImp_Count_6;	(* call FUB R_TRIG *)

	(* reserve counter 7 *)
	xImp_Count_7.CLK 	:= bConnectYourBitToCountHere;					(* change customized *)
	xImp_Count_7;	(* call FUB R_TRIG *)

	(* reserve counter 8 *)
	xImp_Count_8.CLK 	:= bConnectYourBitToCountHere;  				(* change customized *)
	xImp_Count_8;	(* call FUB R_TRIG *)

	(* reserve counter 9 *)
	xImp_Count_9.CLK 	:=  bConnectYourBitToCountHere;					(* change customized *)
	xImp_Count_9;	(* call FUB R_TRIG *)

	(* reserve counter 10 *)
	xImp_Count_10.CLK 	:=  bConnectYourBitToCountHere1;					(* change customized *)
	xImp_Count_10;	(* call FUB R_TRIG *)

	(***********************************************************************)
	(* extended counter items 11- ONLY FOR USE WITH HMI Extension Package! *)
	(***********************************************************************)

	(* reserve counter 11 *)
	xImp_Count_11.CLK 	:=  bConnectYourBitToCountHere;			(* change customized *)
	xImp_Count_11;	(* call FUB R_TRIG *)

	(* reserve counter 12 *)
	xImp_Count_12.CLK 	:=  bConnectYourBitToCountHere;			(* change customized *)
	xImp_Count_12;	(* call FUB R_TRIG *)

	(* reserve counter 13 *)
	xImp_Count_13.CLK 	:=  bConnectYourBitToCountHere;			(* change customized *)
	xImp_Count_13;	(* call FUB R_TRIG *)

	(* reserve counter 14 *)
	xImp_Count_14.CLK 	:=  bConnectYourBitToCountHere;			(* change customized *)
	xImp_Count_14;	(* call FUB R_TRIG *)

	(* reserve counter 15 *)
	xImp_Count_15.CLK 	:=  bConnectYourBitToCountHere;			(* change customized *)
	xImp_Count_15;	(* call FUB R_TRIG *)

	(* reserve counter 16 *)
	xImp_Count_16.CLK 	:=  bConnectYourBitToCountHere;			(* change customized *)
	xImp_Count_16;	(* call FUB R_TRIG *)

	(* reserve counter 17 *)
	xImp_Count_17.CLK 	:=  bConnectYourBitToCountHere;			(* change customized *)
	xImp_Count_17;	(* call FUB R_TRIG *)

	(* reserve counter 18 *)
	xImp_Count_18.CLK 	:=  bConnectYourBitToCountHere;			(* change customized *)
	xImp_Count_18;	(* call FUB R_TRIG *)

	(* reserve counter 19 *)
	xImp_Count_19.CLK 	:=  bConnectYourBitToCountHere;			(* change customized *)
	xImp_Count_19;	(* call FUB R_TRIG *)

	(* reserve counter 20 *)
	//	bOpt_10msTaskClock := TRUE;								(* to activate the msec counter function with iCount20 *)
	xImp_Count_20.CLK 	:=  bConnectYourBitToCountHere;			(* change customized *) (* default prepared for speeed measurement msec counter; can be reused for other tasks, if necessary *)
	xImp_Count_20;	(* call FUB R_TRIG *)
	(*10msTaskClock on iCount20, prepared for transmission speeed measurements; can be reused at any time for other tasks on customer engines *)
	IF bOpt_10msTaskClock THEN
		VIS2MM.iCount20 := VIS2MM.iCount20 + 10;  (*in TC#2*) 	(* cycle counter as msec counter function with bOpt_10msTaskClock *)
		IF (tRealTime.hour = 23 AND  tRealTime.minute = 59) THEN	VIS2MM.iCount10 := 0;	END_IF		(* reset daily at midnight *)
	END_IF

	(* display operating hour counter - for local display needs only, NOT CHANGEABLE HERE *)
	IN_CU.tImp_OpHour.Do;
	IN_CU.iCnt_OpHours;

	(* display start counter - for local needs only, NOT CHANGEABLE HERE  *)
	IN_CU.bImp_Start ;
	IN_CU.iCnt_Starts;

	OUT_CU.bRPM_Count1	:= IN_CU.tImp_OpHour.Do;  (* := bConnectYourBitToStartTimeHere OR IN_CU.bRPM_Count1_Act;		(* change customized *)
	OUT_CU.bRPM_Count2	:= bConnectYourBitToStartTimeHere OR IN_CU.bRPM_Count2_Act;		(* change customized *)
	OUT_CU.bRPM_Count3	:= bConnectYourBitToStartTimeHere OR IN_CU.bRPM_Count3_Act;		(* change customized *)
	OUT_CU.bRPM_Count4	:= bConnectYourBitToStartTimeHere OR IN_CU.bRPM_Count4_Act;		(* change customized *)
	OUT_CU.bRPM_Count5	:= bConnectYourBitToStartTimeHere OR IN_CU.bRPM_Count5_Act;		(* change customized *)
	OUT_CU.bRPM_Count6	:= bConnectYourBitToStartTimeHere OR IN_CU.bRPM_Count6_Act;		(* change customized *)
	OUT_CU.bRPM_Count7	:= bConnectYourBitToStartTimeHere OR IN_CU.bRPM_Count7_Act;		(* change customized *)
	OUT_CU.bRPM_Count8	:= bConnectYourBitToStartTimeHere OR IN_CU.bRPM_Count8_Act;		(* change customized *)
	OUT_CU.bRPM_Count9	:= bConnectYourBitToStartTimeHere OR IN_CU.bRPM_Count9_Act;		(* change customized *)
	OUT_CU.bRPM_Count10	:= bConnectYourBitToStartTimeHere OR IN_CU.bRPM_Count10_Act;		(* change customized *)
	OUT_CU.bRPM_Count11	:= bConnectYourBitToStartTimeHere OR IN_CU.bRPM_Count11_Act;		(* change customized *)
	OUT_CU.bRPM_Count12	:= bConnectYourBitToStartTimeHere OR IN_CU.bRPM_Count12_Act;		(* change customized *)
	OUT_CU.bRPM_Count13	:= bConnectYourBitToStartTimeHere OR IN_CU.bRPM_Count13_Act;		(* change customized *)
	OUT_CU.bRPM_Count14	:= bConnectYourBitToStartTimeHere OR IN_CU.bRPM_Count14_Act;		(* change customized *)
	OUT_CU.bRPM_Count15	:= bConnectYourBitToStartTimeHere OR IN_CU.bRPM_Count15_Act;		(* change customized *)
	OUT_CU.bRPM_Count16	:= bConnectYourBitToStartTimeHere OR IN_CU.bRPM_Count16_Act;		(* change customized *)

	(**********************************************)
	(*****      END OF CONFIGURATION AREA     *****)
	(**********************************************)

	(* evaluation operating hour impulse *)
	h_imp(CLK := IN_CU.tImp_OpHour.Do );
	IF h_imp.Q THEN	(* if an operation hour is finished *)

	(* Allow user inputs to the counter values*)
//	IF NOT bBlockCounter_UserInput THEN
//		IF VIS2MM.iCount1 <> iCount_InputDetect[1] THEN Perm.iCount1 := VIS2MM.iCount1; END_IF		(*detect and process user inputs *)
//		IF VIS2MM.iCount2 <> iCount_InputDetect[2] THEN Perm.iCount2 := VIS2MM.iCount2; END_IF		(*detect and process user inputs *)
//		IF VIS2MM.iCount3 <> iCount_InputDetect[3] THEN Perm.iCount3 := VIS2MM.iCount3; END_IF		(*detect and process user inputs *)
//		IF VIS2MM.iCount4 <> iCount_InputDetect[4] THEN Perm.iCount4 := VIS2MM.iCount4; END_IF		(*detect and process user inputs *)
//
//
//		IF VIS2MM.iMaintenanceCount1 <> iMaintenanceCount_InputDetect[1] THEN Perm.iMaintenanceCount1 := VIS2MM.iMaintenanceCount1; END_IF		(*detect and process user inputs *)
//		IF VIS2MM.iMaintenanceCount2 <> iMaintenanceCount_InputDetect[2] THEN Perm.iMaintenanceCount2 := VIS2MM.iMaintenanceCount2; END_IF		(*detect and process user inputs *)
//		IF VIS2MM.iMaintenanceCount3 <> iMaintenanceCount_InputDetect[3] THEN Perm.iMaintenanceCount3 := VIS2MM.iMaintenanceCount3; END_IF		(*detect and process user inputs *)
//		IF VIS2MM.iMaintenanceCount4 <> iMaintenanceCount_InputDetect[4] THEN Perm.iMaintenanceCount4 := VIS2MM.iMaintenanceCount4; END_IF		(*detect and process user inputs *)
//	END_IF

		(* maintenance counter 1 *)
		VIS2MM.iMaintenanceCount1   := VIS2MM.iMaintenanceCount1 - 1;		(* decrease counter *)
		(* check limits *)
		IF VIS2MM.iMaintenanceCount1 >= 1000000000 THEN
			VIS2MM.iMaintenanceCount1 := VIS2MM.iMaintenanceCount1 - 1000000000;		(* check upper limit *)
		ELSIF VIS2MM.iMaintenanceCount1 <= -1000000000 THEN
			VIS2MM.iMaintenanceCount1 := VIS2MM.iMaintenanceCount1 + 1000000000;		(* check lower limit *)
		END_IF;
//		IF 	OUT_CU.iMaintenanceCount1 <> VIS2MM.iMaintenanceCount1 THEN		(*detect counter change*)
			OUT_CU.iMaintenanceCount1		 := VIS2MM.iMaintenanceCount1;
			MM2VIS.iMaintenanceCount1		 := VIS2MM.iMaintenanceCount1;
//			iMaintenanceCount_InputDetect[1] := VIS2MM.iMaintenanceCount1;
//		END_IF

		(* maintenance counter 2 *)
		VIS2MM.iMaintenanceCount2   := VIS2MM.iMaintenanceCount2 - 1;		(* decrease counter *)
		(* check limits *)
		IF VIS2MM.iMaintenanceCount2 >= 1000000000 THEN
			VIS2MM.iMaintenanceCount2 := VIS2MM.iMaintenanceCount2 - 1000000000;		(* check upper limit *)
		ELSIF VIS2MM.iMaintenanceCount2 <= -1000000000 THEN
			VIS2MM.iMaintenanceCount2 := VIS2MM.iMaintenanceCount2 + 1000000000;		(* check lower limit *)
		END_IF;
//		IF 	OUT_CU.iMaintenanceCount2 <> VIS2MM.iMaintenanceCount2 THEN		(*detect counter change*)
			OUT_CU.iMaintenanceCount2		 := VIS2MM.iMaintenanceCount2;
			MM2VIS.iMaintenanceCount2		 := VIS2MM.iMaintenanceCount2;
//			iMaintenanceCount_InputDetect[2] := VIS2MM.iMaintenanceCount2;
//		END_IF

		(* maintenance counter 3 *)
		VIS2MM.iMaintenanceCount3   := VIS2MM.iMaintenanceCount3 - 1;		(* decrease counter *)
		(* check limits *)
		IF VIS2MM.iMaintenanceCount3 >= 1000000000 THEN
			VIS2MM.iMaintenanceCount3 := VIS2MM.iMaintenanceCount3 - 1000000000;		(* check upper limit *)
		ELSIF VIS2MM.iMaintenanceCount3 <= -1000000000 THEN
			VIS2MM.iMaintenanceCount3 := VIS2MM.iMaintenanceCount3 + 1000000000;		(* check lower limit *)
		END_IF;
//		IF 	OUT_CU.iMaintenanceCount3 <> VIS2MM.iMaintenanceCount3 THEN		(*detect counter change*)
			OUT_CU.iMaintenanceCount3		 := VIS2MM.iMaintenanceCount3;
			MM2VIS.iMaintenanceCount3		 := VIS2MM.iMaintenanceCount3;
//			iMaintenanceCount_InputDetect[3] := VIS2MM.iMaintenanceCount3;
//		END_IF

		(* maintenance counter 4 *)
		VIS2MM.iMaintenanceCount4   := VIS2MM.iMaintenanceCount4 - 1;		(* decrease counter *)
		(* check limits *)
		IF VIS2MM.iMaintenanceCount4 >= 1000000000 THEN
			VIS2MM.iMaintenanceCount4 := VIS2MM.iMaintenanceCount4 - 1000000000;		(* check upper limit *)
		ELSIF VIS2MM.iMaintenanceCount4 <= -1000000000 THEN
			VIS2MM.iMaintenanceCount4 := VIS2MM.iMaintenanceCount4 + 1000000000;		(* check lower limit *)
		END_IF;
//		IF 	OUT_CU.iMaintenanceCount4 <> VIS2MM.iMaintenanceCount4 THEN		(*detect counter change*)
			OUT_CU.iMaintenanceCount4		 := VIS2MM.iMaintenanceCount4;
			MM2VIS.iMaintenanceCount4		 := VIS2MM.iMaintenanceCount4;
//			iMaintenanceCount_InputDetect[4] := VIS2MM.iMaintenanceCount4;
//		END_IF

		(* maintenance counter 5 *)
		VIS2MM.iMaintenanceCount5   := VIS2MM.iMaintenanceCount5 - 1;		(* decrease counter *)
		(* check limits *)
		IF VIS2MM.iMaintenanceCount5 >= 1000000000 THEN
			VIS2MM.iMaintenanceCount5 := VIS2MM.iMaintenanceCount5 - 1000000000;		(* check upper limit *)
		ELSIF VIS2MM.iMaintenanceCount5 <= -1000000000 THEN
			VIS2MM.iMaintenanceCount5 := VIS2MM.iMaintenanceCount5 + 1000000000;		(* check lower limit *)
		END_IF;
		OUT_CU.iMaintenanceCount5		 := VIS2MM.iMaintenanceCount5;
		MM2VIS.iMaintenanceCount5		 := VIS2MM.iMaintenanceCount5;

		(* maintenance counter 6 *)
		VIS2MM.iMaintenanceCount6   := VIS2MM.iMaintenanceCount6 - 1;		(* decrease counter *)
		(* check limits *)
		IF VIS2MM.iMaintenanceCount6 >= 1000000000 THEN
			VIS2MM.iMaintenanceCount6 := VIS2MM.iMaintenanceCount6 - 1000000000;		(* check upper limit *)
		ELSIF VIS2MM.iMaintenanceCount6 <= -1000000000 THEN
			VIS2MM.iMaintenanceCount6 := VIS2MM.iMaintenanceCount6 + 1000000000;		(* check lower limit *)
		END_IF;
		OUT_CU.iMaintenanceCount6		 := VIS2MM.iMaintenanceCount6;
		MM2VIS.iMaintenanceCount6		 := VIS2MM.iMaintenanceCount6;

		(* maintenance counter 7 *)
		VIS2MM.iMaintenanceCount7   := VIS2MM.iMaintenanceCount7 - 1;		(* decrease counter *)
		(* check limits *)
		IF VIS2MM.iMaintenanceCount7 >= 1000000000 THEN
			VIS2MM.iMaintenanceCount7 := VIS2MM.iMaintenanceCount7 - 1000000000;		(* check upper limit *)
		ELSIF VIS2MM.iMaintenanceCount7 <= -1000000000 THEN
			VIS2MM.iMaintenanceCount7 := VIS2MM.iMaintenanceCount7 + 1000000000;		(* check lower limit *)
		END_IF;
		OUT_CU.iMaintenanceCount7		 := VIS2MM.iMaintenanceCount7;
		MM2VIS.iMaintenanceCount7		 := VIS2MM.iMaintenanceCount7;

		(* maintenance counter 8 *)
		VIS2MM.iMaintenanceCount8   := VIS2MM.iMaintenanceCount8 - 1;		(* decrease counter *)
		(* check limits *)
		IF VIS2MM.iMaintenanceCount8 >= 1000000000 THEN
			VIS2MM.iMaintenanceCount8 := VIS2MM.iMaintenanceCount8 - 1000000000;		(* check upper limit *)
		ELSIF VIS2MM.iMaintenanceCount8 <= -1000000000 THEN
			VIS2MM.iMaintenanceCount8 := VIS2MM.iMaintenanceCount8 + 1000000000;		(* check lower limit *)
		END_IF;
		OUT_CU.iMaintenanceCount8		 := VIS2MM.iMaintenanceCount8;
		MM2VIS.iMaintenanceCount8		 := VIS2MM.iMaintenanceCount8;

	END_IF;

	(* evaluation of the maintenance counter *)

	WART := FALSE;	(* prepare evaluation *)
	IF VIS2MM.iMaintenanceCount1 < 1 THEN
		WART := TRUE;		(* group message because of maintenance counter 1 *)
	END_IF;
	IF VIS2MM.iMaintenanceCount2 < 1 THEN
		WART := TRUE;		(* group message because of maintenance counter 2 *)
	END_IF;
	IF VIS2MM.iMaintenanceCount3 < 1 THEN
		WART := TRUE;		(* group message because of maintenance counter 3 *)
	END_IF;
	IF VIS2MM.iMaintenanceCount4 < 1 THEN
		WART := TRUE;		(* group message because of maintenance counter 4 *)
	END_IF;

	IF VIS2MM.iMaintenanceCount5 < 1 THEN
		WART := TRUE;		(* group message because of maintenance counter 51 *)
	END_IF;
	IF VIS2MM.iMaintenanceCount6 < 1 THEN
		WART := TRUE;		(* group message because of maintenance counter 6 *)
	END_IF;
	IF VIS2MM.iMaintenanceCount7 < 1 THEN
		WART := TRUE;		(* group message because of maintenance counter 7 *)
	END_IF;
	IF VIS2MM.iMaintenanceCount8 < 1 THEN
		WART := TRUE;		(* group message because of maintenance counter 8 *)
	END_IF;

	OUT_CU.bReqMaintenance := WART;	(*connect new MM Output bit to trigger warning in MM op_state*)

	(*Predefinition of new added maintenance counters 5-8*)
	IF 	VIS2MM.iMaintenanceCount5 = 0 AND
		VIS2MM.iMaintenanceCount6 = 0 AND
		VIS2MM.iMaintenanceCount7 = 0 AND
		VIS2MM.iMaintenanceCount8 = 0 AND
		IN_CU.iCnt_OpHours 		<= 10 AND					(*V4.10*)
		IN_CU.iCnt_Starts 		<= 10 AND					(*V4.10*)
		IN_CU.tPB2MM.bParaSetupOk
	THEN
		VIS2MM.iMaintenanceCount5 := 500000;
		VIS2MM.iMaintenanceCount6 := 600000;
		VIS2MM.iMaintenanceCount7 := 700000;
		VIS2MM.iMaintenanceCount8 := 800000;
	END_IF

	(* evaluation reserve counter *)

	(* reserve counter 1 *)
	IF xImp_Count_1.Q THEN
		(* increase counter *)
		VIS2MM.iCount1 := VIS2MM.iCount1 + 1;
		(* check limits *)
		IF VIS2MM.iCount1 >= 1000000000 THEN
			VIS2MM.iCount1 := VIS2MM.iCount1 - 1000000000;		(* check upper limit *)
		ELSIF VIS2MM.iCount1 <= -1000000000 THEN
			VIS2MM.iCount1 := VIS2MM.iCount1 + 1000000000;		(* check lower limit *)
		END_IF;
	END_IF;
	OUT_CU.iCount1			:= VIS2MM.iCount1;
	MM2VIS.iCount1			:= VIS2MM.iCount1;

	(* reserve counter 2 *)
	IF xImp_Count_2.Q THEN
		(* increase counter *)
		VIS2MM.iCount2 := VIS2MM.iCount2 + 1;
		(* check limits *)
		IF VIS2MM.iCount2 >= 1000000000 THEN
			VIS2MM.iCount2 := VIS2MM.iCount2 - 1000000000;		(* check upper limit *)
		ELSIF VIS2MM.iCount2 <= -1000000000 THEN
			VIS2MM.iCount2 := VIS2MM.iCount2 + 1000000000;		(* check lower limit *)
		END_IF;
	END_IF;
	OUT_CU.iCount2			:= VIS2MM.iCount2;
	MM2VIS.iCount2			:= VIS2MM.iCount2;

	(* reserve counter 3 *)
	IF xImp_Count_3.Q THEN
		(* increase counter *)
		VIS2MM.iCount3 := VIS2MM.iCount3 + 1;
		(* check limits *)
		IF VIS2MM.iCount3 >= 1000000000 THEN
			VIS2MM.iCount3 := VIS2MM.iCount3 - 1000000000;		(* check upper limit *)
		ELSIF VIS2MM.iCount3 <= -1000000000 THEN
			VIS2MM.iCount3 := VIS2MM.iCount3 + 1000000000;		(* check lower limit *)
		END_IF;
	END_IF;
	OUT_CU.iCount3			:= VIS2MM.iCount3;
	MM2VIS.iCount3			:= VIS2MM.iCount3;

	(* reserve counter 4 *)
	IF xImp_Count_4.Q THEN
		VIS2MM.iCount4 := VIS2MM.iCount4 + 1;
		(* check limits *)
		IF VIS2MM.iCount4 >= 1000000000 THEN
			VIS2MM.iCount4 := VIS2MM.iCount4 - 1000000000;		(* check upper limit *)
		ELSIF VIS2MM.iCount4 <= -1000000000 THEN
			VIS2MM.iCount4 := VIS2MM.iCount4 + 1000000000;		(* check lower limit *)
		END_IF;
	END_IF;
	OUT_CU.iCount4			:= VIS2MM.iCount4;
	MM2VIS.iCount4			:= VIS2MM.iCount4;

	(* reserve counter 5 *)
	IF xImp_Count_5.Q THEN
		(* increase counter *)
		VIS2MM.iCount5 := VIS2MM.iCount5 + 1;
		(* check limits *)
		IF VIS2MM.iCount5 >= 1000000000 THEN
			VIS2MM.iCount5 := VIS2MM.iCount5 - 1000000000;		(* check upper limit *)
		ELSIF VIS2MM.iCount5 <= -1000000000 THEN
			VIS2MM.iCount5 := VIS2MM.iCount5 + 1000000000;		(* check lower limit *)
		END_IF;
	END_IF;
	OUT_CU.iCount5			:= VIS2MM.iCount5;
	MM2VIS.iCount5			:= VIS2MM.iCount5;

	(* reserve counter 6 *)
	IF xImp_Count_6.Q THEN
		(* increase counter *)
		VIS2MM.iCount6 := VIS2MM.iCount6 + 1;
		(* check limits *)
		IF VIS2MM.iCount6 >= 1000000000 THEN
			VIS2MM.iCount6 := VIS2MM.iCount6 - 1000000000;		(* check upper limit *)
		ELSIF VIS2MM.iCount6 <= -1000000000 THEN
			VIS2MM.iCount6 := VIS2MM.iCount6 + 1000000000;		(* check lower limit *)
		END_IF;
	END_IF;
	OUT_CU.iCount6			:= VIS2MM.iCount6;
	MM2VIS.iCount6			:= VIS2MM.iCount6;

	(* reserve counter 7 *)
	IF xImp_Count_7.Q THEN
		(* increase counter *)
		VIS2MM.iCount7 := VIS2MM.iCount7 + 1;
		(* check limits *)
		IF VIS2MM.iCount7 >= 1000000000 THEN
			VIS2MM.iCount7 := VIS2MM.iCount7 - 1000000000;		(* check upper limit *)
		ELSIF VIS2MM.iCount7 <= -1000000000 THEN
			VIS2MM.iCount7 := VIS2MM.iCount7 + 1000000000;		(* check lower limit *)
		END_IF;
	END_IF;
	OUT_CU.iCount7			:= VIS2MM.iCount7;
	MM2VIS.iCount7			:= VIS2MM.iCount7;

	(* reserve counter 8 *)
	IF xImp_Count_8.Q THEN
		(* increase counter *)
		VIS2MM.iCount8 := VIS2MM.iCount8 + 1;
		(* check limits *)
		IF VIS2MM.iCount8 >= 1000000000 THEN
			VIS2MM.iCount8 := VIS2MM.iCount8 - 1000000000;		(* check upper limit *)
		ELSIF VIS2MM.iCount8 <= -1000000000 THEN
			VIS2MM.iCount8 := VIS2MM.iCount8 + 1000000000;		(* check lower limit *)
		END_IF;
	END_IF;
	OUT_CU.iCount8			:= VIS2MM.iCount8;
	MM2VIS.iCount8			:= VIS2MM.iCount8;

	(* reserve counter 9 *)
	IF xImp_Count_9.Q THEN
		(* increase counter *)
		VIS2MM.iCount9 := VIS2MM.iCount9 + 1;
		(* check limits *)
		IF VIS2MM.iCount9 >= 1000000000 THEN
			VIS2MM.iCount9 := VIS2MM.iCount9 - 1000000000;		(* check upper limit *)
		ELSIF VIS2MM.iCount9 <= -1000000000 THEN
			VIS2MM.iCount9 := VIS2MM.iCount9 + 1000000000;		(* check lower limit *)
		END_IF;
	END_IF;
	OUT_CU.iCount9			:= VIS2MM.iCount9;
	MM2VIS.iCount9			:= VIS2MM.iCount9;

	(* reserve counter 10 *)
	IF xImp_Count_10.Q THEN
		(* increase counter *)
		VIS2MM.iCount10 := VIS2MM.iCount10 + 1;
		(* check limits *)
		IF VIS2MM.iCount10 >= 1000000000 THEN
			VIS2MM.iCount10 := VIS2MM.iCount10 - 1000000000;		(* check upper limit *)
		ELSIF VIS2MM.iCount10 <= -1000000000 THEN
			VIS2MM.iCount10 := VIS2MM.iCount10 + 1000000000;		(* check lower limit *)
		END_IF;
	END_IF;
	OUT_CU.iCount10			:= VIS2MM.iCount10;
	MM2VIS.iCount10			:= VIS2MM.iCount10;

	(* reserve counter 11 *)
	IF xImp_Count_11.Q THEN
		(* increase counter *)
		VIS2MM.iCount11 := VIS2MM.iCount11 + 1;
		(* check limits *)
		IF VIS2MM.iCount11 >= 1000000000 THEN
			VIS2MM.iCount11 := VIS2MM.iCount11 - 1000000000;		(* check upper limit *)
		ELSIF VIS2MM.iCount11 <= -1000000000 THEN
			VIS2MM.iCount11 := VIS2MM.iCount11 + 1000000000;		(* check lower limit *)
		END_IF;
	END_IF;
	OUT_CU.iCount11			:= VIS2MM.iCount11;
	MM2VIS.iCount11			:= VIS2MM.iCount11;

	(* reserve counter 12 *)
	IF xImp_Count_12.Q THEN
		(* increase counter *)
		VIS2MM.iCount12 := VIS2MM.iCount12 + 1;
		(* check limits *)
		IF VIS2MM.iCount12 >= 1000000000 THEN
			VIS2MM.iCount12 := VIS2MM.iCount12 - 1000000000;		(* check upper limit *)
		ELSIF VIS2MM.iCount12 <= -1000000000 THEN
			VIS2MM.iCount12 := VIS2MM.iCount12 + 1000000000;		(* check lower limit *)
		END_IF;
	END_IF;
	OUT_CU.iCount12			:= VIS2MM.iCount12;
	MM2VIS.iCount12			:= VIS2MM.iCount12;

	(* reserve counter 13 *)
	IF xImp_Count_13.Q THEN
		(* increase counter *)
		VIS2MM.iCount13 := VIS2MM.iCount13 + 1;
		(* check limits *)
		IF VIS2MM.iCount13 >= 1000000000 THEN
			VIS2MM.iCount13 := VIS2MM.iCount13 - 1000000000;		(* check upper limit *)
		ELSIF VIS2MM.iCount13 <= -1000000000 THEN
			VIS2MM.iCount13 := VIS2MM.iCount13 + 1000000000;		(* check lower limit *)
		END_IF;
	END_IF;
	OUT_CU.iCount13			:= VIS2MM.iCount13;
	MM2VIS.iCount13			:= VIS2MM.iCount13;

	(* reserve counter 14 *)
	IF xImp_Count_14.Q THEN
		(* increase counter *)
		VIS2MM.iCount14 := VIS2MM.iCount14 + 1;
		(* check limits *)
		IF VIS2MM.iCount14 >= 1000000000 THEN
			VIS2MM.iCount14 := VIS2MM.iCount14 - 1000000000;		(* check upper limit *)
		ELSIF VIS2MM.iCount14 <= -1000000000 THEN
			VIS2MM.iCount14 := VIS2MM.iCount14 + 1000000000;		(* check lower limit *)
		END_IF;
	END_IF;
	OUT_CU.iCount14			:= VIS2MM.iCount14;
	MM2VIS.iCount14			:= VIS2MM.iCount14;

	(* reserve counter 15 *)
	IF xImp_Count_15.Q THEN
		(* increase counter *)
		VIS2MM.iCount15 := VIS2MM.iCount15 + 1;
		(* check limits *)
		IF VIS2MM.iCount15 >= 1000000000 THEN
			VIS2MM.iCount15 := VIS2MM.iCount15 - 1000000000;		(* check upper limit *)
		ELSIF VIS2MM.iCount15 <= -1000000000 THEN
			VIS2MM.iCount15 := VIS2MM.iCount15 + 1000000000;		(* check lower limit *)
		END_IF;
	END_IF;
	OUT_CU.iCount15			:= VIS2MM.iCount15;
	MM2VIS.iCount15			:= VIS2MM.iCount15;

	(* reserve counter 16 *)
	IF xImp_Count_16.Q THEN
		(* increase counter *)
		VIS2MM.iCount16 := VIS2MM.iCount16 + 1;
		(* check limits *)
		IF VIS2MM.iCount16 >= 1000000000 THEN
			VIS2MM.iCount16 := VIS2MM.iCount16 - 1000000000;		(* check upper limit *)
		ELSIF VIS2MM.iCount16 <= -1000000000 THEN
			VIS2MM.iCount16 := VIS2MM.iCount16 + 1000000000;		(* check lower limit *)
		END_IF;
	END_IF;
	OUT_CU.iCount16			:= VIS2MM.iCount16;
	MM2VIS.iCount16			:= VIS2MM.iCount16;

	(* reserve counter 17 *)
	IF xImp_Count_17.Q THEN
		(* increase counter *)
		VIS2MM.iCount17 := VIS2MM.iCount17 + 1;
		(* check limits *)
		IF VIS2MM.iCount17 >= 1000000000 THEN
			VIS2MM.iCount17 := VIS2MM.iCount17 - 1000000000;		(* check upper limit *)
		ELSIF VIS2MM.iCount17 <= -1000000000 THEN
			VIS2MM.iCount17 := VIS2MM.iCount17 + 1000000000;		(* check lower limit *)
		END_IF;
	END_IF;
	OUT_CU.iCount17			:= VIS2MM.iCount17;
	MM2VIS.iCount17			:= VIS2MM.iCount17;

	(* reserve counter 18 *)
	IF xImp_Count_18.Q THEN
		(* increase counter *)
		VIS2MM.iCount18 := VIS2MM.iCount18 + 1;
		(* check limits *)
		IF VIS2MM.iCount18 >= 1000000000 THEN
			VIS2MM.iCount18 := VIS2MM.iCount18 - 1000000000;		(* check upper limit *)
		ELSIF VIS2MM.iCount18 <= -1000000000 THEN
			VIS2MM.iCount18 := VIS2MM.iCount18 + 1000000000;		(* check lower limit *)
		END_IF;
	END_IF;
	OUT_CU.iCount18			:= VIS2MM.iCount18;
	MM2VIS.iCount18			:= VIS2MM.iCount18;

	(* reserve counter 19 *)
	IF xImp_Count_19.Q THEN
		(* increase counter *)
		VIS2MM.iCount19 := VIS2MM.iCount19 + 1;
		(* check limits *)
		IF VIS2MM.iCount19 >= 1000000000 THEN
			VIS2MM.iCount19 := VIS2MM.iCount19 - 1000000000;		(* check upper limit *)
		ELSIF VIS2MM.iCount19 <= -1000000000 THEN
			VIS2MM.iCount19 := VIS2MM.iCount19 + 1000000000;		(* check lower limit *)
		END_IF;
	END_IF;
	OUT_CU.iCount19			:= VIS2MM.iCount19;
	MM2VIS.iCount19			:= VIS2MM.iCount19;

	(* reserve counter 20 *)
	IF xImp_Count_20.Q THEN
		(* increase counter *)
		VIS2MM.iCount20 := VIS2MM.iCount20 + 1;
		(* check limits *)
		IF VIS2MM.iCount20 >= 1000000000 THEN
			VIS2MM.iCount20 := VIS2MM.iCount20 - 1000000000;		(* check upper limit *)
		ELSIF VIS2MM.iCount20 <= -1000000000 THEN
			VIS2MM.iCount20 := VIS2MM.iCount20 + 1000000000;		(* check lower limit *)
		END_IF;
	END_IF;
	OUT_CU.iCount20			:= VIS2MM.iCount20;
	MM2VIS.iCount20			:= VIS2MM.iCount20;

	(* evaluation of the RPM counter *)

	IF tRealTime.second <> real_old THEN	(* duration once every second *)
		real_old := tRealTime.second;

		IF OUT_CU.iRPS_h = 0 THEN  		(* at 00:00 (RPS) reset of the counters *)
			IF OUT_CU.iRPS_m = 0 THEN
				reset := TRUE;
			END_IF;
		ELSE
			reset := FALSE;
		END_IF;

		(* time step 10 sec *)
		treset.IN := reset;
		treset.PT := t#10s;

		treset;  (* call FUB TP *)

		resetrpm := treset.Q;
		tresetrpm.CLK := resetrpm;

		tresetrpm; (* call FUB R_TRIG *)

		IF tresetrpm.Q THEN (* reset counters *)
			MM2VIS.tRPM_Count1.count  := 0;
			MM2VIS.tRPM_Count2.count  := 0;
			MM2VIS.tRPM_Count3.count  := 0;
			MM2VIS.tRPM_Count4.count  := 0;
			MM2VIS.tRPM_Count5.count  := 0;
			MM2VIS.tRPM_Count6.count  := 0;
			MM2VIS.tRPM_Count7.count  := 0;
			MM2VIS.tRPM_Count8.count  := 0;
			MM2VIS.tRPM_Count9.count  := 0;
			MM2VIS.tRPM_Count10.count := 0;
			MM2VIS.tRPM_Count11.count := 0;
			MM2VIS.tRPM_Count12.count := 0;
			MM2VIS.tRPM_Count13.count := 0;
			MM2VIS.tRPM_Count14.count := 0;
			MM2VIS.tRPM_Count15.count := 0;
			MM2VIS.tRPM_Count16.count := 0;
		END_IF;

		IF OUT_CU.bRPM_Count1 THEN		(* report time measuring 1 *)
			MM2VIS.tRPM_Count1.count := MM2VIS.tRPM_Count1.count + 1;
			IF  NOT resetrpm THEN
				MM2VIS.tRPM_Count1.h := DINT_TO_INT(MM2VIS.tRPM_Count1.count / 3600);
				MM2VIS.tRPM_Count1.m := DINT_TO_INT((MM2VIS.tRPM_Count1.count MOD 3600) / 60);
				MM2VIS.tRPM_Count1.s := DINT_TO_INT(MM2VIS.tRPM_Count1.count MOD 60);
			END_IF;
		END_IF;

		IF OUT_CU.bRPM_Count2 THEN		(* report time measuring 2 *)
			MM2VIS.tRPM_Count2.count := MM2VIS.tRPM_Count2.count + 1;
			IF NOT resetrpm THEN
				MM2VIS.tRPM_Count2.h := DINT_TO_INT(MM2VIS.tRPM_Count2.count / 3600);
				MM2VIS.tRPM_Count2.m := DINT_TO_INT((MM2VIS.tRPM_Count2.count MOD 3600) / 60);
				MM2VIS.tRPM_Count2.s := DINT_TO_INT(MM2VIS.tRPM_Count2.count MOD 60);
			END_IF;
		END_IF;

		IF OUT_CU.bRPM_Count3 THEN		(* report time measuring 3 *)
			MM2VIS.tRPM_Count3.count := MM2VIS.tRPM_Count3.count + 1;
			IF NOT resetrpm THEN
				MM2VIS.tRPM_Count3.h := DINT_TO_INT(MM2VIS.tRPM_Count3.count / 3600);
				MM2VIS.tRPM_Count3.m := DINT_TO_INT((MM2VIS.tRPM_Count3.count MOD 3600) / 60);
				MM2VIS.tRPM_Count3.s := DINT_TO_INT(MM2VIS.tRPM_Count3.count MOD 60);
			END_IF;
		END_IF;

		IF OUT_CU.bRPM_Count4 THEN		(* report time measuring 4 *)
			MM2VIS.tRPM_Count4.count := MM2VIS.tRPM_Count4.count + 1;
			IF  NOT resetrpm  THEN
				MM2VIS.tRPM_Count4.h := DINT_TO_INT(MM2VIS.tRPM_Count4.count / 3600);
				MM2VIS.tRPM_Count4.m := DINT_TO_INT((MM2VIS.tRPM_Count4.count MOD 3600) / 60);
				MM2VIS.tRPM_Count4.s := DINT_TO_INT(MM2VIS.tRPM_Count4.count MOD 60);
			END_IF;
		END_IF;

		IF OUT_CU.bRPM_Count5 THEN		(* report time measuring 5 *)
			MM2VIS.tRPM_Count5.count := MM2VIS.tRPM_Count5.count + 1;
			IF NOT resetrpm THEN
				MM2VIS.tRPM_Count5.h := DINT_TO_INT(MM2VIS.tRPM_Count5.count / 3600);
				MM2VIS.tRPM_Count5.m := DINT_TO_INT((MM2VIS.tRPM_Count5.count MOD 3600) / 60);
				MM2VIS.tRPM_Count5.s := DINT_TO_INT(MM2VIS.tRPM_Count5.count MOD 60);
			END_IF;
		END_IF;

		IF OUT_CU.bRPM_Count6 THEN		(* report time measuring 6 *)
			MM2VIS.tRPM_Count6.count := MM2VIS.tRPM_Count6.count + 1;
			IF NOT resetrpm THEN
				MM2VIS.tRPM_Count6.h := DINT_TO_INT(MM2VIS.tRPM_Count6.count / 3600);
				MM2VIS.tRPM_Count6.m := DINT_TO_INT((MM2VIS.tRPM_Count6.count MOD 3600) / 60);
				MM2VIS.tRPM_Count6.s := DINT_TO_INT(MM2VIS.tRPM_Count6.count MOD 60);
			END_IF;
		END_IF;

		IF OUT_CU.bRPM_Count7 THEN		(* report time measuring 7 *)
			MM2VIS.tRPM_Count7.count := MM2VIS.tRPM_Count7.count + 1;
			IF  NOT resetrpm THEN
				MM2VIS.tRPM_Count7.h := DINT_TO_INT(MM2VIS.tRPM_Count7.count / 3600);
				MM2VIS.tRPM_Count7.m := DINT_TO_INT((MM2VIS.tRPM_Count7.count MOD 3600) / 60);
				MM2VIS.tRPM_Count7.s := DINT_TO_INT(MM2VIS.tRPM_Count7.count MOD 60);
			END_IF;
		END_IF;

		IF OUT_CU.bRPM_Count8 THEN		(* report time measuring 8 *)
			MM2VIS.tRPM_Count8.count := MM2VIS.tRPM_Count8.count + 1;
			IF  NOT resetrpm THEN
				MM2VIS.tRPM_Count8.h := DINT_TO_INT(MM2VIS.tRPM_Count8.count / 3600);
				MM2VIS.tRPM_Count8.m := DINT_TO_INT((MM2VIS.tRPM_Count8.count MOD 3600) / 60);
				MM2VIS.tRPM_Count8.s := DINT_TO_INT(MM2VIS.tRPM_Count8.count MOD 60);
			END_IF;
		END_IF;

		IF OUT_CU.bRPM_Count9 THEN		(* report time measuring 9 *)
			MM2VIS.tRPM_Count9.count := MM2VIS.tRPM_Count9.count + 1;
			IF NOT resetrpm THEN
				MM2VIS.tRPM_Count9.h := DINT_TO_INT(MM2VIS.tRPM_Count9.count / 3600);
				MM2VIS.tRPM_Count9.m := DINT_TO_INT((MM2VIS.tRPM_Count9.count MOD 3600) / 60);
				MM2VIS.tRPM_Count9.s := DINT_TO_INT(MM2VIS.tRPM_Count9.count MOD 60);
			END_IF;
		END_IF;

		IF OUT_CU.bRPM_Count10 THEN		(* report time measuring 10 *)
			MM2VIS.tRPM_Count10.count := MM2VIS.tRPM_Count10.count + 1;
			IF NOT resetrpm THEN
				MM2VIS.tRPM_Count10.h := DINT_TO_INT(MM2VIS.tRPM_Count10.count / 3600);
				MM2VIS.tRPM_Count10.m := DINT_TO_INT((MM2VIS.tRPM_Count10.count MOD 3600) / 60);
				MM2VIS.tRPM_Count10.s := DINT_TO_INT(MM2VIS.tRPM_Count10.count MOD 60);
			END_IF;
		END_IF;

		IF OUT_CU.bRPM_Count11 THEN		(* report time measuring 11 *)
			MM2VIS.tRPM_Count11.count := MM2VIS.tRPM_Count11.count + 1;
			IF NOT resetrpm THEN
				MM2VIS.tRPM_Count11.h := DINT_TO_INT(MM2VIS.tRPM_Count11.count / 3600);
				MM2VIS.tRPM_Count11.m := DINT_TO_INT((MM2VIS.tRPM_Count11.count MOD 3600) / 60);
				MM2VIS.tRPM_Count11.s := DINT_TO_INT(MM2VIS.tRPM_Count11.count MOD 60);
			END_IF;
		END_IF;

		IF OUT_CU.bRPM_Count12 THEN		(* report time measuring 12 *)
			MM2VIS.tRPM_Count12.count := MM2VIS.tRPM_Count12.count + 1;
			IF  NOT resetrpm THEN
				MM2VIS.tRPM_Count12.h := DINT_TO_INT(MM2VIS.tRPM_Count12.count / 3600);
				MM2VIS.tRPM_Count12.m := DINT_TO_INT((MM2VIS.tRPM_Count12.count MOD 3600) / 60);
				MM2VIS.tRPM_Count12.s := DINT_TO_INT(MM2VIS.tRPM_Count12.count MOD 60);
			END_IF;
		END_IF;

		IF OUT_CU.bRPM_Count13 THEN		(* report time measuring 13 *)
			MM2VIS.tRPM_Count13.count := MM2VIS.tRPM_Count13.count + 1;
			IF NOT resetrpm THEN
				MM2VIS.tRPM_Count13.h := DINT_TO_INT(MM2VIS.tRPM_Count13.count / 3600);
				MM2VIS.tRPM_Count13.m := DINT_TO_INT((MM2VIS.tRPM_Count13.count MOD 3600) / 60);
				MM2VIS.tRPM_Count13.s := DINT_TO_INT(MM2VIS.tRPM_Count13.count MOD 60);
			END_IF;
		END_IF;

		IF OUT_CU.bRPM_Count14 THEN		(* report time measuring 14 *)
			MM2VIS.tRPM_Count14.count := MM2VIS.tRPM_Count14.count + 1;
			IF NOT resetrpm THEN
				MM2VIS.tRPM_Count14.h := DINT_TO_INT(MM2VIS.tRPM_Count14.count / 3600);
				MM2VIS.tRPM_Count14.m := DINT_TO_INT((MM2VIS.tRPM_Count14.count MOD 3600) / 60);
				MM2VIS.tRPM_Count14.s := DINT_TO_INT(MM2VIS.tRPM_Count14.count MOD 60);
			END_IF;
		END_IF;

		IF OUT_CU.bRPM_Count15 THEN		(* report time measuring 15 *)
			MM2VIS.tRPM_Count15.count := MM2VIS.tRPM_Count15.count + 1;
			IF NOT resetrpm THEN
				MM2VIS.tRPM_Count15.h := DINT_TO_INT(MM2VIS.tRPM_Count15.count / 3600);
				MM2VIS.tRPM_Count15.m := DINT_TO_INT((MM2VIS.tRPM_Count15.count MOD 3600) / 60);
				MM2VIS.tRPM_Count15.s := DINT_TO_INT(MM2VIS.tRPM_Count15.count MOD 60);
			END_IF;
		END_IF;

		IF OUT_CU.bRPM_Count16 THEN		(* report time measuring 16 *)
			MM2VIS.tRPM_Count16.count := MM2VIS.tRPM_Count16.count + 1;
			IF NOT resetrpm THEN
				MM2VIS.tRPM_Count16.h := DINT_TO_INT(MM2VIS.tRPM_Count16.count / 3600);
				MM2VIS.tRPM_Count16.m := DINT_TO_INT((MM2VIS.tRPM_Count16.count MOD 3600) / 60);
				MM2VIS.tRPM_Count16.s := DINT_TO_INT(MM2VIS.tRPM_Count16.count MOD 60);
			END_IF;
		END_IF;

	END_IF;

	(********************************************************************************)
	(* setting date and time														*)
	(* The visual display system sets the new time and date						    *)
	(* At the transition of bSetClock form TRUE to FALSE the real time clock of the *)
	(* PLC is set to the date and time form the visual display system				*)

// TIME SET NICHT MEHR NOTWENDIG?
//	F_TRIG_GetTime(CLK:=bGetWinClock);			(* trigger to falling edge of dia.ne win time set *)
//	IF bSetClock OR (F_TRIG_GetTime.Q AND NOT bWinFail) THEN
//
//		IF bSetClock THEN
//			tSetTime.year := 2000 + RPS_JAHR2;
//			RPS_JAHR      := tSetTime.year;
//		ELSE
//			tSetTime.year := RPS_JAHR;
//			RPS_JAHR2     := tSetTime.year - 2000;
//		END_IF;
//		tSetTime.month 	:= UINT_TO_USINT(OUT_CU.iRPS_Month);
//		tSetTime.day	:= UINT_TO_USINT(OUT_CU.iRPS_Day);
//		tSetTime.hour	:= UINT_TO_USINT(OUT_CU.iRPS_h);
//		tSetTime.minute	:= UINT_TO_USINT(OUT_CU.iRPS_m);
//		tSetTime.second	:= UINT_TO_USINT(OUT_CU.iRPS_s);
//
//		(* setting time of the controller *)
//		DTExSetTime_RPS.DT1 := DTStructure_TO_DT(ADR(tSetTime));	(* change format *)
//		DTExSetTime_RPS(enable:=1, DT1:=DTExSetTime_RPS.DT1, Option:= timEXSETTIME_NO_LOGENTRY); (* setting *)
//
//	END_IF;
	bWinFail := FALSE;		(* reset WIN failure bit *)

	(* getting time of the controller *)

	DTGetTime_RPS(enable:=1);		(* getting *)
	DT_TO_DTStructure(DTGetTime_RPS.DT1, ADR(tRealTime));		(* change format *)

	(* generate one tick for each second and one tick for each minute 	*)
	(* tick duration is one cycle of task class 3 (= 100 ms)			*)
	IF tRealTime.second <> ucLastSecond THEN		(* second tick *)
		ucLastSecond := tRealTime.second;
		bSecondTick := TRUE;
		IF tRealTime.minute <> ucLastMinute THEN	(* minute tick *)
			ucLastMinute := tRealTime.minute;
			bMinuteTick := TRUE;
		ELSE
			bMinuteTick := FALSE;
		END_IF;
	ELSE
		bSecondTick := FALSE;
	END_IF;

//	(* get clock from DIA.NE WIN every minute *)
//
//	IF bWinServerOn AND OUT_CU.iRPS_s = 30 THEN
//		bGetWinClock  := TRUE;
//	END_IF;
//
//	TON_WinAlive.IN := bGetWinClock OR usSetWinClock = usWinSetValue;
//	TON_WinAlive.PT := T#5s;
//	TON_WinAlive;
//	IF TON_WinAlive.Q THEN
//		bGetWinClock  := FALSE;
//		usSetWinClock := 0;
//		bWinFail      := TRUE;		(* no time change because WIN did not answer within 5 seconds *)
//	END_IF;

//	(* setting DIA.NE WIN clock if pannel clock will be set *)
//
//	IF EDGENEG(bSetClock) THEN
//		usSetWinClock := usWinSetValue;
//	END_IF;

	(* read clock from panel controller *)

//	IF bSecondTick AND NOT bSetClock AND usSetWinClock <> usWinSetValue AND NOT bGetWinClock THEN		(* processing every one second *)
//
//		(* preparation of the RPS time *)
//		RPS_JAHR	:= tRealTime.year;
//		RPS_JAHR2   := RPS_JAHR - 2000; (* for visualising only last 2 digits on the display*)
//		OUT_CU.iRPS_Month		:= tRealTime.month;
//		OUT_CU.iRPS_Day		:= tRealTime.day;
//		RPS_WOTAG	:= tRealTime.reserve;
//		OUT_CU.iRPS_h		:= tRealTime.hour;
//		OUT_CU.iRPS_m		:= tRealTime.minute;
//		OUT_CU.iRPS_s		:= tRealTime.second;
//
//	END_IF; 		(* end of processing every one second *)

//	(* preparation of the RPS time *)
//
//	ulRPSTime := ADR(ucRPSTime);

	(* end program *)

	(* Task outputs *)
		OUT_CU.iCount1;
		OUT_CU.iCount2;
		OUT_CU.iCount3;
		OUT_CU.iCount4;

		OUT_CU.iCount5;
		OUT_CU.iCount6;
		OUT_CU.iCount7;
		OUT_CU.iCount8;
		OUT_CU.iCount9;
		OUT_CU.iCount10;

		OUT_CU.iCount11;
		OUT_CU.iCount12;
		OUT_CU.iCount13;
		OUT_CU.iCount14;
		OUT_CU.iCount15;
		OUT_CU.iCount16;
		OUT_CU.iCount17;
		OUT_CU.iCount18;
		OUT_CU.iCount19;
		OUT_CU.iCount20;

		OUT_CU.iMaintenanceCount1;
		OUT_CU.iMaintenanceCount2;
		OUT_CU.iMaintenanceCount3;
		OUT_CU.iMaintenanceCount4;

		OUT_CU.iMaintenanceCount5;
		OUT_CU.iMaintenanceCount6;
		OUT_CU.iMaintenanceCount7;
		OUT_CU.iMaintenanceCount8;

		OUT_CU.iRPS_Month;		(*obsolete?*)
		OUT_CU.iRPS_Day;		(*obsolete?*)
		OUT_CU.iRPS_h	;		(*obsolete?*)
		OUT_CU.iRPS_m	;		(*obsolete?*)
		OUT_CU.iRPS_s	;		(*obsolete?*)

END_PROGRAM
```

#### counterInit.st
```iecst
(*******************************************************************************
AGGR: counter.st - connection and processing of counters (init)

This code is confidential and proprietary to the INNIO Company.
It may not be used in any form, or reproduced in any manner, without the express
written permission of the INNIO Company.
Copyright, INNIO Company, 2019

- set actual software version of engine controller

Customized modifications: -
------------------------

History:
-------
V0.1	05-03-2002	Weitzer, generated from zaehler.c / V0.1
...
V3.20	03-11-2010	Weitzer, change to version 3.20

Instructions for use:
--------------------

!! Task MOVED TO op_state!!

Outstandings:
------------

*******************************************************************************)

PROGRAM _INIT
	(*Predefinition of new added maintenance counters 5-8*)
	IF 	VIS2MM.iMaintenanceCount5 = 0 AND
		VIS2MM.iMaintenanceCount6 = 0 AND
		VIS2MM.iMaintenanceCount7 = 0 AND
		VIS2MM.iMaintenanceCount8 = 0
	THEN
		VIS2MM.iMaintenanceCount5 := 500000;
		VIS2MM.iMaintenanceCount6 := 600000;
		VIS2MM.iMaintenanceCount7 := 700000;
		VIS2MM.iMaintenanceCount8 := 800000;
	END_IF

	(* set actual software version of engine controller *)
//	prog_vers := 390;	(*Set displayed PLC version number here*)  (* ?ALT? *)

	(* global tags for other task *)
//	ucCodeComplete;  	(* wer hat das angelegt? wofür? *)
//	bLogOK;				(* wer hat das angelegt? wofür? *)
//	usVisTempID;		(* wer hat das angelegt? wofür? *)
//	ulTempID;			(* wer hat das angelegt? wofür? *)

END_PROGRAM
```

#### counter.var
```iecst
VAR
	bMinuteTick : BOOL; (* TRUE for 0,1s if one min. is over *)
	bSecondTick : BOOL; (* TRUE for 0,1s if one sec. is over *)
	reset : BOOL; (* reset at 00:00 *)
	resetrpm : BOOL; (* reset RPM *)
	h_imp : R_TRIG;
	xImp_Count_1 : R_TRIG; (* R_TRIG structure counter 1 *)
	xImp_Count_2 : R_TRIG; (* R_TRIG structure counter 2 *)
	xImp_Count_3 : R_TRIG; (* R_TRIG structure counter 3 *)
	xImp_Count_4 : R_TRIG; (* R_TRIG structure counter 4 *)
	xImp_Count_5 : R_TRIG; (* R_TRIG structure counter 5*)
	xImp_Count_6 : R_TRIG; (* R_TRIG structure counter 6*)
	xImp_Count_7 : R_TRIG; (* R_TRIG structure counter 7*)
	xImp_Count_8 : R_TRIG; (* R_TRIG structure counter 8*)
	xImp_Count_9 : R_TRIG; (* R_TRIG structure counter 9*)
	xImp_Count_10 : R_TRIG; (* R_TRIG structure counter 10*)
	xImp_Count_11 : R_TRIG; (* R_TRIG structure counter 11*)
	xImp_Count_12 : R_TRIG; (* R_TRIG structure counter 12*)
	xImp_Count_13 : R_TRIG; (* R_TRIG structure counter 13*)
	xImp_Count_14 : R_TRIG; (* R_TRIG structure counter 14*)
	xImp_Count_15 : R_TRIG; (* R_TRIG structure counter 15*)
	xImp_Count_16 : R_TRIG; (* R_TRIG structure counter 16*)
	xImp_Count_17 : R_TRIG; (* R_TRIG structure counter 17*)
	xImp_Count_18 : R_TRIG; (* R_TRIG structure counter 18*)
	xImp_Count_19 : R_TRIG; (* R_TRIG structure counter 19*)
	xImp_Count_20 : R_TRIG; (* R_TRIG structure counter 20*)
	tresetrpm : R_TRIG; (* R_TRIG structure time reset RPM *)
	treset : TP; (* TP structure time reset *)
	real_old : UINT; (* save old real time second *)
	ucLastSecond : USINT;
	ucLastMinute : USINT;
	DTGetTime_RPS : DTGetTime;
	bWinFail : BOOL;
	bConnectYourBitToCountHere1 : BOOL := FALSE; (*replace this placeholder with customized value*)
	bConnectYourBitToCountHere2 : BOOL := FALSE; (*replace this placeholder with customized value*)
	bConnectYourBitToCountHere3 : BOOL := FALSE; (*replace this placeholder with customized value*)
	bConnectYourBitToCountHere4 : BOOL := FALSE; (*replace this placeholder with customized value*)
	bConnectYourBitToCountHere : BOOL := FALSE; (*replace this placeholder with customized value*)
	bConnectYourBitToStartTimeHere : BOOL; (*Placeholder for local variable*)
	WART : BOOL;
	bOpt_10msTaskClock : BOOL := FALSE; (*SET TO FALSE, if iCount20 is used for customized functions. TRUE activates default function: msec counter*)
END_VAR
```
